(*Sensori di extra corsa + home + tastatori + presenza elemento nella pinza*)
MachinePalletizerModules.AX_X.IN.Px_Touch_1			 		:= Ok_sensores_Tastator OR (Re_In_TastatorePinza[1]  AND Re_In_TastatorePinza[2]) ;
MachinePalletizerModules.AX_X.IN.Px_Touch_2			 		:= Ok_sensores_Tastator OR ( Re_In_TastatorePinza[3]  AND Re_In_TastatorePinza[4]) ;
//MachinePalletizerModules.AX_X.IN.PX_TouchEmergency_1		:= I_TastatoreEmergenzaPinza_1 AND I_TastatoreEmergenzaPinza_2 AND I_TastatoreEmergenzaPinza_3 AND I_TastatoreEmergenzaPinza_4 OR NOT TouchErrorEnable;
MachinePalletizerModules.AX_X.IN.PX_TouchEmergency_1		:= (Re_In_TastatoreEmergenzaPinza[1] AND Re_In_TastatoreEmergenzaPinza[2])OR NOT TouchErrorEnable;
MachinePalletizerModules.AX_X.IN.PX_TouchEmergency_2		:= (Re_In_TastatoreEmergenzaPinza[3] AND Re_In_TastatoreEmergenzaPinza[4])OR NOT TouchErrorEnable;
MachinePalletizerModules.AX_X.IN.PX_GripPresence			:= NOT I_PHPresenzaMaterialePinza;
MachinePalletizerModules.AX_X.IN.Enable_TouchEmergency   	:= ADR(TouchErrorEnable);

MachinePalletizerModules.AX_X.Ax^.PxNegative 			:= NOT I_ExtraCorsaNegativo_X ;
MachinePalletizerModules.AX_X.Ax^.PxPositive 			:= NOT I_ExtraCorsaPositivo_X ;
IF MachinePalletizerModules.AX_X.AxHomingParameters^.InvertiDirezione THEN
	MachinePalletizerModules.AX_X.Ax^.PxHome 			:= NOT I_ExtraCorsaPositivo_X;
ELSE
	MachinePalletizerModules.AX_X.Ax^.PxHome 			:= NOT I_ExtraCorsaNegativo_X;
END_IF

MachinePalletizerModules.AX_X.Ax^.PxNegativeEnable 		:= TRUE;
MachinePalletizerModules.AX_X.Ax^.PxPositiveEnable 		:= TRUE;
MachinePalletizerModules.AX_X.Ax^.HomeExecutedAlwaysOn 	:= TRUE;
MachinePalletizerModules.AX_X.Ax^.DriveNeedReset 		:= DriveNeedReset;

MachinePalletizerModules.AX_X.Ax^.Parameter.MAXPosition 			:= AxisPar_X.MaxPosition;
MachinePalletizerModules.AX_X.Ax^.Parameter.MinPosition 			:= AxisPar_X.MinPosition;
MachinePalletizerModules.AX_X.Ax^.Parameter.HomeLagError			:= 0;
MachinePalletizerModules.AX_X.Ax^.EnableAutoWritePositionLimit 		:= TRUE;
(* Varie Modulo*)
MachinePalletizerModules.AX_X.AxisPar 					:= ADR(AxisPar_X);
MachinePalletizerModules.AX_X.ManCmd					:= ADR(ManCmd.X);
MachinePalletizerModules.AX_X.Cfg.TimeBase 				:= TimeBase;
MachinePalletizerModules.AX_X.Programma					:= ADR(ProgrammaToModule_X);


//@@@@@@@@@@@@@@@@@@@@@@@@@@@@@@@@@@@@@@@@@@@@@@@@@@@@@@@@@@@@@@@@@@@@@@@@@@@@@@@
ProgramaEjes.EjeX := ProgrammaToModule_X.ID ;
ProgramaEjes.CoordenadaEjeX := ProgrammaToModule_X.Quota_Destinazione ;
//@@@@@@@@@@@@@@@@@@@@@@@@@@@@@@@@@@@@@@@@@@@@@@@@@@@@@@@@@@@@@@@@@@@@@@@@@@@@@@
EncoderEsternoAsse_X.Pronto								:= I_EncoderX_Pronto;
MachinePalletizerModules.AX_X.EncoderEsterno			:= ADR(EncoderEsternoAsse_X);

(*AGGIORNAMENTO STATO DEL PROGEMMA IN ESECUZIONE*)
Programma_X[ProgrammaToModule_X.ID].Stato := ProgrammaToModule_X.Stato;
(************************************************************************
******************************* MODULO Y ********************************
************************************************************************)
(* Configurazione Asse Y *)
MachinePalletizerModules.AX_Y.Ax 							:= ADR(Y_AxisLib);
MachinePalletizerModules.AX_Y.Ax^.AxRef 					:= ADR(Y_Axis);
MachinePalletizerModules.AX_Y.Ax^.TimeBase 					:= TimeBase;
MachinePalletizerModules.AX_Y.Ax^.PowerEnable 				:= PowerEnableAssi;
MachinePalletizerModules.AX_Y.Ax^.PowerEnablePositive    	:= PowerEnableAssi AND (I_ExtraCorsaPositivo_Y OR NOT TouchErrorEnable);
MachinePalletizerModules.AX_Y.Ax^.PowerEnableNegative    	:= PowerEnableAssi AND (I_ExtraCorsaNegativo_Y OR NOT TouchErrorEnable);
MachinePalletizerModules.AX_Y.Ax^.EncoderType				:= ABSOLUTE_ENCODER;
MachinePalletizerModules.AX_Y.AxHomingParameters			:= ADR(AxisHomingParameters_Y);

(*Sensori di extra corsa + home + tastatori + presenza elemento nella pinza + sicurezza cinghia*)
MachinePalletizerModules.AX_Y.IN.BeltSafety				:= I_SicurezzaCinghia_Y OR NOT TouchErrorEnable;
MachinePalletizerModules.AX_Y.IN.Px_Touch_1			 	:= Ok_sensores_Tastator OR (Re_In_TastatorePinza[1]  AND Re_In_TastatorePinza[2]) ;
MachinePalletizerModules.AX_Y.IN.Px_Touch_2			 	:= Ok_sensores_Tastator OR (Re_In_TastatorePinza[3]  AND Re_In_TastatorePinza[4]) ;
//MachinePalletizerModules.AX_Y.IN.PX_TouchEmergency_1		:= I_TastatoreEmergenzaPinza_1 AND I_TastatoreEmergenzaPinza_2 AND I_TastatoreEmergenzaPinza_3 AND I_TastatoreEmergenzaPinza_4 OR NOT TouchErrorEnable;
MachinePalletizerModules.AX_Y.IN.PX_TouchEmergency_1		:= (Re_In_TastatoreEmergenzaPinza[1] AND Re_In_TastatoreEmergenzaPinza[2]) OR NOT TouchErrorEnable;
MachinePalletizerModules.AX_Y.IN.PX_TouchEmergency_2		:= ( Re_In_TastatoreEmergenzaPinza[3] AND Re_In_TastatoreEmergenzaPinza[4] )OR NOT TouchErrorEnable;;
MachinePalletizerModules.AX_Y.IN.PX_GripPresence			:= NOT I_PHPresenzaMaterialePinza;
MachinePalletizerModules.AX_Y.IN.Enable_TouchEmergency   := ADR(TouchErrorEnable);
MachinePalletizerModules.AX_Y.IN.SimulazioneSenzaHW		:= FALSE;//TEST_ENABLE;
MachinePalletizerModules.AX_Y.AbilitaOffsetInUscitaTasteggio   := TRUE;//FROM_HMI_PAL.HMI_AbilitaOffsetUscitaTasteggioPrelPallet;
MachinePalletizerModules.AX_Y.OffsetUscitaDaTasteggio	:=  HMI_OffsetUscitaTastatori;
MachinePalletizerModules.AX_Y.VelocitaDiUscitaDaTastatori := HMI_VelocitaDiUscitaDaTastatoriAxY;

MachinePalletizerModules.AX_Y.Ax^.PxNegative 			:= NOT I_ExtraCorsaNegativo_Y;
MachinePalletizerModules.AX_Y.Ax^.PxPositive 			:= NOT I_ExtraCorsaPositivo_Y;

IF MachinePalletizerModules.AX_Y.AxHomingParameters^.InvertiDirezione THEN
	MachinePalletizerModules.AX_Y.Ax^.PxHome 			:= NOT I_ExtraCorsaPositivo_Y;
ELSE
	MachinePalletizerModules.AX_Y.Ax^.PxHome 			:= NOT I_ExtraCorsaNegativo_Y;
END_IF

(* Varie Modulo*)
MachinePalletizerModules.AX_Y.Ax^.PxNegativeEnable 		:= TRUE;
MachinePalletizerModules.AX_Y.Ax^.PxPositiveEnable 		:= TRUE;
MachinePalletizerModules.AX_Y.Ax^.HomeExecutedAlwaysOn 	:= TRUE;
MachinePalletizerModules.AX_Y.Ax^.DriveNeedReset 		:= DriveNeedReset;

MachinePalletizerModules.AX_Y.Ax^.Parameter.MAXPosition 			:= AxisPar_Y.MaxPosition;
MachinePalletizerModules.AX_Y.Ax^.Parameter.MinPosition 			:= AxisPar_Y.MinPosition;
MachinePalletizerModules.AX_Y.Ax^.EnableAutoWritePositionLimit 		:= TRUE;
MachinePalletizerModules.AX_Y.Ax^.Parameter.HomeLagError			:= 0;

MachinePalletizerModules.AX_Y.AxisPar 					:= ADR(AxisPar_Y);
//MachinePalletizerModules.AX_Y.Status 					:= ADR(Status);
MachinePalletizerModules.AX_Y.ManCmd					:= ADR(ManCmd.Y);
MachinePalletizerModules.AX_Y.Cfg.TimeBase 				:= TimeBase;
MachinePalletizerModules.AX_Y.Programma					:= ADR(ProgrammaToModule_Y);

//@@@@@@@@@@@@@@@@@@@@@@@@@@@@@@@@@@@@@@@@@@@@@@@@@@@@@@@@@@
ProgramaEjes.EjeY := ProgrammaToModule_Y.ID;
ProgramaEjes.CoordenadaEjeY := ProgrammaToModule_Y.Quota_Destinazione;
//@@@@@@@@@@@@@@@@@@@@@@@@@@@@@@@@@@@@@@@@@@@@@@@@@@@@@@@@@@

//MachinePalletizerModules.AX_Y.ProgrammaNEXT				:= ADR(ProgrammaToModuleNEXT_Y);
(*AGGIORNAMENTO STATO DEL PROGEMMA IN ESECUZIONE*)
Programma_Y[ProgrammaToModule_Y.ID].Stato := ProgrammaToModule_Y.Stato;
//Programma_Y[ProgrammaToModuleNEXT_Y.ID].Stato := ProgrammaToModuleNEXT_Y.Stato;
(************************************************************************
******************************* MODULO Z ********************************
************************************************************************)
(* Configurazione Asse Z *)
MachinePalletizerModules.AX_Z.Ax 						:= ADR(Z_AxisLib);
MachinePalletizerModules.AX_Z.Ax^.AxRef 					:= ADR(Z_Axis);
MachinePalletizerModules.AX_Z.Ax^.TimeBase 				:= TimeBase;
MachinePalletizerModules.AX_Z.Ax^.PowerEnable 			:= PowerEnableAssi;
MachinePalletizerModules.AX_Z.Ax^.PowerEnablePositive    := PowerEnableAssi AND (I_ExtraCorsaPositivo_Z OR NOT TouchErrorEnable)AND (I_FermoSicurezzaRilasciato OR I_StartCicloPal);
//MachinePalletizerModules.AX_Z.Ax^.PowerEnableNegative    := PowerEnableAssi AND (I_ExtraCorsaNegativo_Z AND (I_TastatoreEmergenzaPinza_1 AND I_TastatoreEmergenzaPinza_2) OR NOT TouchErrorEnable) AND (I_FermoSicurezzaRilasciato OR I_StartCicloPal);
MachinePalletizerModules.AX_Z.Ax^.PowerEnableNegative    := PowerEnableAssi 
																AND (I_ExtraCorsaNegativo_Z AND (Re_In_TastatoreEmergenzaPinza[1] AND Re_In_TastatoreEmergenzaPinza[1]) 
																			OR NOT TouchErrorEnable) AND (I_FermoSicurezzaRilasciato OR I_StartCicloPal);
MachinePalletizerModules.AX_Z.Ax^.EncoderType			:= ABSOLUTE_ENCODER;
MachinePalletizerModules.AX_Z.AxHomingParameters			:= ADR(AxisHomingParameters_Z);

MachinePalletizerModules.AX_Z.Ax^.BrakePresent := false;//TRUE;
MachinePalletizerModules.AX_Z.Ax^.BrakeEnable  := FALSE;//TRUE;
MachinePalletizerModules.AX_Z.Ax^.Parameter.TimeBrakeOff := 200;
MachinePalletizerModules.AX_Z.Ax^.Parameter.TimeBrakeOn  := 200;
MachinePalletizerModules.AX_Z.Ax^.Parameter.TimeBrakeActivation := 60000;


(*Sensori di extra corsa + home + tastatori + presenza elemento nella pinza + sicurezza cinghia*)
MachinePalletizerModules.AX_Z.IN.BeltSafety				:= I_SicurezzaCinghia_Z OR NOT TouchErrorEnable;	

(* Gestione dei tastatori in base al tipo di prelievo ovvero all'elemento che è presente in prelievo *)
MachinePalletizerModules.AX_Z.ByPassTastatoriInUscitaTasteggio 	:= FALSE;
MachinePalletizerModules.AX_Z.InterventoPxASpazio				:= FALSE;
MachinePalletizerModules.AX_Z.SpazioInteventoPX					:= HMI_SpazioInterventoTastoriCartone;

MachinePalletizerModules.AX_Z.IN.Px_Touch_1			 		:= Ok_sensores_Tastator OR (Re_In_TastatorePinza[1]  AND Re_In_TastatorePinza[2]) ;
MachinePalletizerModules.AX_Z.IN.Px_Touch_2			 		:= Ok_sensores_Tastator OR (Re_In_TastatorePinza[3]  AND Re_In_TastatorePinza[4]) ;
//MachinePalletizerModules.AX_Z.IN.PX_TouchEmergency_1		:= I_TastatoreEmergenzaPinza_1 AND I_TastatoreEmergenzaPinza_2 AND I_TastatoreEmergenzaPinza_3 AND I_TastatoreEmergenzaPinza_4 OR NOT TouchErrorEnable;
MachinePalletizerModules.AX_Z.IN.PX_TouchEmergency_1		:= (Re_In_TastatoreEmergenzaPinza[1] AND Re_In_TastatoreEmergenzaPinza[2] ) OR NOT TouchErrorEnable;
MachinePalletizerModules.AX_Z.IN.PX_TouchEmergency_2		:= (Re_In_TastatoreEmergenzaPinza[3] AND Re_In_TastatoreEmergenzaPinza[4]) OR NOT TouchErrorEnable;;
MachinePalletizerModules.AX_Z.IN.PX_GripPresence			:= NOT I_PHPresenzaMaterialePinza;
MachinePalletizerModules.AX_Z.IN.Enable_TouchEmergency   	:= ADR(TouchErrorEnable);
MachinePalletizerModules.AX_Z.IN.SimulazioneSenzaHW			:= FALSE;//TEST_ENABLE;
(* Gestione Tasteggio *)
MachinePalletizerModules.AX_Z.AbilitaOffsetInUscitaTasteggio   := TRUE;//FROM_HMI_PAL.HMI_AbilitaOffsetUscitaTasteggioPrelPallet;
MachinePalletizerModules.AX_Z.OffsetUscitaDaTasteggio		:= HMI_OffsetUscitaTastatori;
MachinePalletizerModules.AX_Z.VelocitaDiUscitaDaTastatori 	:= HMI_VelocitaDiUscitaDaTastatoriAxZ;
MachinePalletizerModules.AX_Z.TempoRisalitaTastatori 		:= HMI_TempoPresaPiastrella;

MachinePalletizerModules.AX_Z.Ax^.PxNegative 			:= NOT I_ExtraCorsaNegativo_Z;
MachinePalletizerModules.AX_Z.Ax^.PxPositive 			:= NOT I_ExtraCorsaPositivo_Z;
IF MachinePalletizerModules.AX_Z.AxHomingParameters^.InvertiDirezione THEN
	MachinePalletizerModules.AX_Z.Ax^.PxHome 				:= NOT I_ExtraCorsaPositivo_Z;
ELSE
	MachinePalletizerModules.AX_Z.Ax^.PxHome 				:= NOT I_ExtraCorsaNegativo_Z;
END_IF
(* Varie Modulo*)
MachinePalletizerModules.AX_Z.Ax^.PxNegativeEnable 		:= TRUE;//NOT TEST_ENABLE;
MachinePalletizerModules.AX_Z.Ax^.PxPositiveEnable 		:= TRUE;//NOT TEST_ENABLE;
MachinePalletizerModules.AX_Z.Ax^.HomeExecutedAlwaysOn 	:= TRUE;
MachinePalletizerModules.AX_Z.Ax^.DriveNeedReset 		:= DriveNeedReset;//NOT TEST_ENABLE;

MachinePalletizerModules.AX_Z.Ax^.Parameter.HomeInvertDirection 	:= TRUE;
MachinePalletizerModules.AX_Z.Ax^.Parameter.MAXPosition 			:= AxisPar_Z.MaxPosition;
MachinePalletizerModules.AX_Z.Ax^.Parameter.MinPosition 			:= AxisPar_Z.MinPosition;
MachinePalletizerModules.AX_Z.Ax^.EnableAutoWritePositionLimit 	:= TRUE;
MachinePalletizerModules.AX_Z.Ax^.Parameter.HomeLagError			:= 0;

MachinePalletizerModules.AX_Z.AxisPar 					:= ADR(AxisPar_Z);
//MachinePalletizerModules.AX_Z.Status 					:= ADR(Status);
MachinePalletizerModules.AX_Z.ManCmd						:= ADR(ManCmd.Z);
MachinePalletizerModules.AX_Z.Cfg.TimeBase 				:= TimeBase;
MachinePalletizerModules.AX_Z.Programma					:= ADR(ProgrammaToModule_Z);
//@@@@@@@@@@@@@@@@@@@@@@@@@@@@@@@@@@@@@@@@@@@@@@@@@@@@@@@@@@
ProgramaEjes.EjeZ := ProgrammaToModule_Z.ID;
ProgramaEjes.CoordenadaEjeZ := ProgrammaToModule_Z.Quota_Destinazione;
//@@@@@@@@@@@@@@@@@@@@@@@@@@@@@@@@@@@@@@@@@@@@@@@@@@@@@@@@@@

//MachinePalletizerModules.AX_Z.ProgrammaNEXT				:= ADR(ProgrammaToModuleNEXT_Z);

(*AGGIORNAMENTO STATO DEL PROGEMMA IN ESECUZIONE*)
Programma_Z[ProgrammaToModule_Z.ID].Stato := ProgrammaToModule_Z.Stato;
//Programma_Z[ProgrammaToModuleNEXT_Z.ID].Stato := ProgrammaToModuleNEXT_Z.Stato;

(************************************************************************
******************************* MODULO J ********************************
************************************************************************)
(* Configurazione Asse J *)
MachinePalletizerModules.AX_J.Ax 						:= ADR(J_AxisLib);
MachinePalletizerModules.AX_J.Ax^.AxRef 				:= ADR(J_Axis);
MachinePalletizerModules.AX_J.Ax^.TimeBase 				:= TimeBase;
MachinePalletizerModules.AX_J.AxisPar 					:= ADR(AxisPar_J);
//MachinePalletizerModules.AX_J.Status 					:= ADR(Status);
MachinePalletizerModules.AX_J.ManCmd					:= ADR(ManCmd.J);
MachinePalletizerModules.AX_J.Cfg.TimeBase 				:= TimeBase;
MachinePalletizerModules.AX_J.Programma					:= ADR(ProgrammaToModule_J);
//@@@@@@@@@@@@@@@@@@@@@@@@@@@@@@@@@@@@@@@@@@@@@@@@@@@@@@@@@@
ProgramaEjes.EjeJ := ProgrammaToModule_J.ID;
ProgramaEjes.CoordenadaEjeJ := ProgrammaToModule_J.Quota_Destinazione;

//@@@@@@@@@@@@@@@@@@@@@@@@@@@@@@@@@@@@@@@@@@@@@@@@@@@@@@@@@@
(*RetardoAlarTastatore(IN := NOT I_TastatoreEmergenzaPinza_1 OR NOT I_TastatoreEmergenzaPinza_2 
							OR NOT I_TastatoreEmergenzaPinza_3 OR NOT I_TastatoreEmergenzaPinza_4 ,Pt:=T#30MS);*)
							
							

(*Sensori di extra corsa + home + tastatori + presenza elemento nella pinza*)
MachinePalletizerModules.AX_J.IN.Px_Touch_1			 	:=  Ok_sensores_Tastator OR (Re_In_TastatorePinza[1]  AND Re_In_TastatorePinza[2]) ;
MachinePalletizerModules.AX_J.IN.Px_Touch_2			 	:=  Ok_sensores_Tastator OR (Re_In_TastatorePinza[3]  AND Re_In_TastatorePinza[4]) ;
MachinePalletizerModules.AX_J.IN.PX_TouchEmergency_1	:= (Re_In_TastatoreEmergenzaPinza[1] AND Re_In_TastatoreEmergenzaPinza[2] ) OR NOT TouchErrorEnable;
MachinePalletizerModules.AX_J.IN.PX_TouchEmergency_2	:= (Re_In_TastatoreEmergenzaPinza[3] AND Re_In_TastatoreEmergenzaPinza[4] ) OR NOT TouchErrorEnable;;
MachinePalletizerModules.AX_J.AxHomingParameters		:= ADR(AxisHomingParameters_J);
MachinePalletizerModules.AX_J.Ax^.EncoderType			:= ABSOLUTE_ENCODER;
                                                        
MachinePalletizerModules.AX_J.IN.PX_GripPresence		:= NOT I_PHPresenzaMaterialePinza;
MachinePalletizerModules.AX_J.IN.Enable_TouchEmergency  := ADR(TouchErrorEnable);
MachinePalletizerModules.AX_J.IN.SimulazioneSenzaHW		:= FALSE;//TEST_ENABLE;

MachinePalletizerModules.AX_J.Ax^.TimeBase 				:= TimeBase;
MachinePalletizerModules.AX_J.Ax^.PowerEnable 			:= PowerEnableAssi;
MachinePalletizerModules.AX_J.Ax^.Parameter.HomeInvertDirection 	:= MachinePalletizerModules.AX_J.AxHomingParameters^.InvertiDirezione;
IF MachinePalletizerModules.AX_J.AxHomingParameters^.InvertiDirezione THEN
	MachinePalletizerModules.AX_J.Ax^.PxHome 			:= NOT I_ExtraCorsaPositivo_J;
ELSE
	MachinePalletizerModules.AX_J.Ax^.PxHome 			:= NOT I_ExtraCorsaNegativo_J;
END_IF
MachinePalletizerModules.AX_J.Ax^.PxNegative 			:= NOT I_ExtraCorsaNegativo_J;
MachinePalletizerModules.AX_J.Ax^.PxPositive 			:= NOT I_ExtraCorsaPositivo_J;

MachinePalletizerModules.AX_J.Ax^.PowerEnablePositive    := PowerEnableAssi AND (I_ExtraCorsaPositivo_J OR NOT TouchErrorEnable);
MachinePalletizerModules.AX_J.Ax^.PowerEnableNegative    := PowerEnableAssi AND (I_ExtraCorsaNegativo_J OR NOT TouchErrorEnable);

(* Varie Modulo*)
MachinePalletizerModules.AX_J.Ax^.PxNegativeEnable 		:= TRUE;
MachinePalletizerModules.AX_J.Ax^.PxPositiveEnable 		:= TRUE;//NOT TEST_ENABLE;
MachinePalletizerModules.AX_J.Ax^.HomeExecutedAlwaysOn 	:= TRUE;
MachinePalletizerModules.AX_J.Ax^.DriveNeedReset 		:= DriveNeedReset;//NOT TEST_ENABLE;

MachinePalletizerModules.AX_J.Ax^.Parameter.MAXPosition 			:= AxisPar_J.MaxPosition;
MachinePalletizerModules.AX_J.Ax^.Parameter.MinPosition 			:= AxisPar_J.MinPosition;
MachinePalletizerModules.AX_J.Ax^.EnableAutoWritePositionLimit 		:= TRUE;
MachinePalletizerModules.AX_J.Ax^.Parameter.HomeLagError			:= 0;
//FTC TASTEGGIO
MachinePalletizerModules.AX_J.IN_Pinza.InKeyence0_Byte0		:= I_Keyence180_Byte0;
MachinePalletizerModules.AX_J.IN_Pinza.InKeyence0_Byte1		:= I_Keyence180_Byte1;
MachinePalletizerModules.AX_J.IN_Pinza.InKeyence180_Byte0	:= I_Keyence0_Byte0; 
MachinePalletizerModules.AX_J.IN_Pinza.InKeyence180_Byte1	:= I_Keyence0_Byte1;

(*AGGIORNAMENTO STATO DEL PROGEMMA IN ESECUZIONE*)
Programma_J[ProgrammaToModule_J.ID].Stato := ProgrammaToModule_J.Stato;

{region " PINZA "}
(************************************************************************
***************** MODULO PINZA CON GESTIONE ASPIRAZIONI VARIE *************************
************************************************************************)
MachinePalletizerModules.Pinza.IN.TastoreCartoneDX	 			:= I_TastoreCartone1;
MachinePalletizerModules.Pinza.IN.TastoreCartoneSX	 			:= I_TastoreCartone2;
MachinePalletizerModules.Pinza.IN.ExtraCorsaPinzaSganciata 		:= I_ExtraCorsaPinzaSganciata;
MachinePalletizerModules.Pinza.IN.InKeyence0_Byte0				:= I_Keyence0_Byte0;
MachinePalletizerModules.Pinza.IN.InKeyence0_Byte1				:= I_Keyence0_Byte1;
MachinePalletizerModules.Pinza.IN.InKeyence180_Byte0			:= I_Keyence180_Byte0; 
MachinePalletizerModules.Pinza.IN.InKeyence180_Byte1			:= I_Keyence180_Byte1;

MachinePalletizerModules.Pinza.IN.InKeyence0_Byte0_2			:= I_Keyence0_Byte0_2;
MachinePalletizerModules.Pinza.IN.InKeyence0_Byte1_2			:= I_Keyence0_Byte1_2;
MachinePalletizerModules.Pinza.IN.InKeyence180_Byte0_2			:= I_Keyence180_Byte0_2; 
MachinePalletizerModules.Pinza.IN.InKeyence180_Byte1_2			:= I_Keyence180_Byte1_2;
			   
MachinePalletizerModules.Pinza.ManCmd							:= ADR(ManCmd.Pinza);
MachinePalletizerModules.Pinza.Cfg.TimeBase 					:= TimeBase;
MachinePalletizerModules.Pinza.ModuleJ							:= ADR(MachinePalletizerModules.AX_J);
MachinePalletizerModules.Pinza.Mission							:= ADR(Mission);

(* Cilindro Apertura *)
MachinePalletizerModules.Pinza.CilindroApertura 									:= ADR(CilindroAperturaPinza);
MachinePalletizerModules.Pinza.CilindroApertura^.Enable_RUN 						:= EnablePneumatica;	
MachinePalletizerModules.Pinza.CilindroApertura^.Config.ForceActive_OnStartup 		:= FALSE;				// Se a Startup il cilindro è in stato non definito forza Inattivo (CONFIG)	
MachinePalletizerModules.Pinza.CilindroApertura^.Config.ForceInactive_OnStartup 	:= TRUE;				// Se a Startup il cilindro è in stato non definito forza Attivo (CONFIG)
MachinePalletizerModules.Pinza.CilindroApertura^.Config.TimeBase 					:= Timebase;							// Base dei tempi
MachinePalletizerModules.Pinza.CilindroApertura^.Parameter.ActivationTime 			:= 100;						// [ms] di Attivazione/Timeout (PARAMETRO)
MachinePalletizerModules.Pinza.CilindroApertura^.Parameter.DeactivationTime 		:= 100;						// [ms] di Disattivazione/Timeout (PARAMETRO)
MachinePalletizerModules.Pinza.CilindroApertura^.Parameter.FeedbackType 			:= DEVICE_WITHOUT_FEEDBACK; 	// Scelta dei reed presenti
MachinePalletizerModules.Pinza.CilindroApertura^.Parameter.PxActive_FilterTime_OFF 	:= 0;					// [ms] di filtro sensore Attivo ON (0=NO filtro) (PARAMETRO)
MachinePalletizerModules.Pinza.CilindroApertura^.Parameter.PxActive_FilterTime_ON 	:= 0;					// [ms] di filtro sensore Attivo OFF (0=NO filtro) (PARAMETRO)
MachinePalletizerModules.Pinza.CilindroApertura^.Parameter.PxInactive_FilterTime_OFF 	:= 0;				// [ms] di filtro sensore Inattivo ON (0=NO filtro) (PARAMETRO)
MachinePalletizerModules.Pinza.CilindroApertura^.Parameter.PxInactive_FilterTime_ON 	:= 0;				// [ms] di filtro sensore Inattivo ON (0=NO filtro) (PARAMETRO)
MachinePalletizerModules.Pinza.CilindroApertura^.Parameter.PxLatchFunction_Enable 	:= TRUE;				// Enable gestione sensori con latch (PARAMETRO)
MachinePalletizerModules.Pinza.CilindroApertura^.IN.PX_Active 						:= I_PinzaApertaDX AND I_PinzaApertaSX;	// IN sensore aperto
MachinePalletizerModules.Pinza.CilindroApertura^.IN.PX_Inactive 					:= I_PinzaChiusaDX AND I_PinzaChiusaSX; // IN sensore chiuso	
MachinePalletizerModules.Pinza.IN.FTC_FaldaDX										:= I_PHPresenzaFaldaDX;
MachinePalletizerModules.Pinza.IN.FTC_FaldaSX										:= I_PHPresenzaFaldaSX;
MachinePalletizerModules.Pinza.AbilitaAperturaAutomaticaPinza						:= HMI_AbilitaAperturaAutomaticaPinza;
			   
(* OVEM ventose DX *)	
MachinePalletizerModules.Pinza.AspirazioneDX1 							:= ADR(Ovem1);
MachinePalletizerModules.Pinza.AspirazioneDX1^.IN.LivelloDepressione 	:=  (SHL(I_LivelloDepressioneOVEM_BH_1,8) OR I_LivelloDepressioneOVEM_BL_1) ;
(* Ingressi Ovem *)
MachinePalletizerModules.Pinza.AspirazioneDX1^.IN.PortQualifier		:=  I_PortQualifierOVEM_1;
MachinePalletizerModules.Pinza.AspirazioneDX1^.IN.TimeStamp			:=  I_TimeStampCiabattaPinzaK515;
MachinePalletizerModules.Pinza.AspirazioneDX1^.IN.AirOK				:=  I_AriaOK;
(* Comunicazione OVEM *)
ComunicazioneOvem1.sNetId 												:= F_CreateAmsNetId(I_CiabattaPinzaK515AMSADDR.netId);
ComunicazioneOvem1.nSlaveAddr 											:= I_CiabattaPinzaK515AMSADDR.port;
ComunicazioneOvem1.nPorta 												:= 1;
MachinePalletizerModules.Pinza.AspirazioneDX1^.IN_Comunication			:= ADR(ComunicazioneOvem1);
(* COMANDI *)
MachinePalletizerModules.Pinza.AspirazioneDX1^.Command					:= ADR(CommandOVEM_1);
(* PARAMETRI *)
FROM_HMI_PAL.HMI_OvemParameters.SogliaDepressione_1B 	:= FROM_HMI_PAL.HMI_OvemParameters.SogliaDepressione_1;
FROM_HMI_PAL.HMI_OvemParameters.SogliaDepressione_2 	:= FROM_HMI_PAL.HMI_OvemParameters.SogliaDepressione_1;
FROM_HMI_PAL.HMI_OvemParameters.SogliaDepressione_2B 	:= FROM_HMI_PAL.HMI_OvemParameters.SogliaDepressione_1;
IF (FROM_HMI_PAL.HMI_OvemParameters.SogliaDepressione_1 - FROM_HMI_PAL.HMI_OvemParameters.IsteresiDepressione_1) <= 0 THEN //Se l'isteresi è >= della soglia, la forzo a zero
	FROM_HMI_PAL.HMI_OvemParameters.IsteresiDepressione_1 := 0;
END_IF

MachinePalletizerModules.Pinza.AspirazioneDX1^.Parameters.TempoInvioComandiCoe					:= 40;
MachinePalletizerModules.Pinza.AspirazioneDX1^.IN_TargetParameters								:= FROM_HMI_PAL.HMI_OvemParameters;
MachinePalletizerModules.Pinza.AspirazioneDX1^.Parameters.AbilitaScritturaAutomaticaParametri 	:= TRUE;
MachinePalletizerModules.Pinza.AspirazioneDX1^.Parameters.UtilizzaStatoDepressione_OVEM 		:= TRUE;
MachinePalletizerModules.Pinza.AspirazioneDX1^.Parameters.TimeDepLOST						:= 200;
MachinePalletizerModules.Pinza.AspirazioneDX1^.Parameters.TimeDepOK							:= 100;
MachinePalletizerModules.Pinza.AspirazioneDX1^.Parameters.TipoSoffio							:= 1;//Soffio Automatico e gestito dall'ovem
MachinePalletizerModules.Pinza.AspirazioneDX1^.Parameters.AbilitaCalcoloAutoSoglia			:= TRUE;
MachinePalletizerModules.Pinza.AspirazioneDX1^.Parameters.TipologiaOvem						:= 1;//Ovem di tipo NO
(* OVEM ventose SX *)
MachinePalletizerModules.Pinza.AspirazioneSX1 							:= ADR(Ovem2);
MachinePalletizerModules.Pinza.AspirazioneSX1^.IN.LivelloDepressione 	:=  (SHL(I_LivelloDepressioneOVEM_BH_2,8) OR I_LivelloDepressioneOVEM_BL_2) ;
(* Ingressi Ovem *)
MachinePalletizerModules.Pinza.AspirazioneSX1^.IN.PortQualifier		:=  I_PortQualifierOVEM_2;
MachinePalletizerModules.Pinza.AspirazioneSX1^.IN.TimeStamp			:=  I_TimeStampCiabattaPinzaK516;
MachinePalletizerModules.Pinza.AspirazioneSX1^.IN.AirOK				:=  I_AriaOK;
(* Comunicazione OVEM *)
ComunicazioneOvem2.sNetId 													:= F_CreateAmsNetId(I_CiabattaPinzaK516AMSADDR.netId);
ComunicazioneOvem2.nSlaveAddr 												:= I_CiabattaPinzaK516AMSADDR.port;
ComunicazioneOvem2.nPorta 													:= 1;
MachinePalletizerModules.Pinza.AspirazioneSX1^.IN_Comunication			:= ADR(ComunicazioneOvem2);
(* COMANDI *)
MachinePalletizerModules.Pinza.AspirazioneSX1^.Command					:= ADR(CommandOVEM_2);
(* PARAMETRI *)
MachinePalletizerModules.Pinza.AspirazioneSX1^.Parameters := MachinePalletizerModules.Pinza.AspirazioneDX1^.Parameters;
MachinePalletizerModules.Pinza.AspirazioneSX1^.IN_TargetParameters := MachinePalletizerModules.Pinza.AspirazioneDX1^.IN_TargetParameters;

(* OVEM ventose DX2 *)	
MachinePalletizerModules.Pinza.AspirazioneDX2 							:= ADR(Ovem12);
MachinePalletizerModules.Pinza.AspirazioneDX2^.IN.LivelloDepressione 	:=  (SHL(I_LivelloDepressioneOVEM_BH_12,8) OR I_LivelloDepressioneOVEM_BL_12) ;
(* Ingressi Ovem *)
MachinePalletizerModules.Pinza.AspirazioneDX2^.IN.PortQualifier			:=  I_PortQualifierOVEM_12;
MachinePalletizerModules.Pinza.AspirazioneDX2^.IN.TimeStamp				:=  I_TimeStampCiabattaPinzaK515;
MachinePalletizerModules.Pinza.AspirazioneDX2^.IN.AirOK					:=  I_AriaOK;
(* Comunicazione OVEM *)
ComunicazioneOvem12.sNetId 												:= F_CreateAmsNetId(I_CiabattaPinzaK515AMSADDR.netId);
ComunicazioneOvem12.nSlaveAddr 											:= I_CiabattaPinzaK515AMSADDR.port;
ComunicazioneOvem12.nPorta 												:= 5;
MachinePalletizerModules.Pinza.AspirazioneDX2^.IN_Comunication			:= ADR(ComunicazioneOvem12);
(* COMANDI *)
MachinePalletizerModules.Pinza.AspirazioneDX2^.Command					:= ADR(CommandOVEM_12);
(* PARAMETRI *)
MachinePalletizerModules.Pinza.AspirazioneDX2^.Parameters 			:= MachinePalletizerModules.Pinza.AspirazioneDX1^.Parameters;
MachinePalletizerModules.Pinza.AspirazioneDX2^.IN_TargetParameters 	:= MachinePalletizerModules.Pinza.AspirazioneDX1^.IN_TargetParameters;

(* OVEM ventose SX2 *)
MachinePalletizerModules.Pinza.AspirazioneSX2 							:= ADR(Ovem22);
MachinePalletizerModules.Pinza.AspirazioneSX2^.IN.LivelloDepressione 	:=  (SHL(I_LivelloDepressioneOVEM_BH_22,8) OR I_LivelloDepressioneOVEM_BL_22) ;
(* Ingressi Ovem *)
MachinePalletizerModules.Pinza.AspirazioneSX2^.IN.PortQualifier		:=  I_PortQualifierOVEM_22;
MachinePalletizerModules.Pinza.AspirazioneSX2^.IN.TimeStamp			:=  I_TimeStampCiabattaPinzaK516;
MachinePalletizerModules.Pinza.AspirazioneSX2^.IN.AirOK				:=  I_AriaOK;
(* Comunicazione OVEM *)
ComunicazioneOvem22.sNetId 													:= F_CreateAmsNetId(I_CiabattaPinzaK516AMSADDR.netId);
ComunicazioneOvem22.nSlaveAddr 												:= I_CiabattaPinzaK516AMSADDR.port;
ComunicazioneOvem22.nPorta 													:= 2;
MachinePalletizerModules.Pinza.AspirazioneSX2^.IN_Comunication			:= ADR(ComunicazioneOvem22);
(* COMANDI *)
MachinePalletizerModules.Pinza.AspirazioneSX2^.Command					:= ADR(CommandOVEM_22);
(* PARAMETRI *)
MachinePalletizerModules.Pinza.AspirazioneSX2^.Parameters 			:= MachinePalletizerModules.Pinza.AspirazioneDX1^.Parameters;
MachinePalletizerModules.Pinza.AspirazioneSX2^.IN_TargetParameters 	:= MachinePalletizerModules.Pinza.AspirazioneDX1^.IN_TargetParameters;
						 
MachinePalletizerModules.Pinza.IN.ByPassSensoreVuoto := HMI_AbilitaSimulazioneAVuoto;

(* Cilindro Sblocco Pinza *)
MachinePalletizerModules.Pinza.CilindroSbloccoRotazione 									:= ADR(CilindroSbloccoPinza);
MachinePalletizerModules.Pinza.CilindroSbloccoRotazione^.Enable_RUN 						:= EnablePneumatica;	
MachinePalletizerModules.Pinza.CilindroSbloccoRotazione^.Config.ForceActive_OnStartup 		:= FALSE;				// Se a Startup il cilindro è in stato non definito forza Inattivo (CONFIG)	
MachinePalletizerModules.Pinza.CilindroSbloccoRotazione^.Config.ForceInactive_OnStartup 	:= TRUE;				// Se a Startup il cilindro è in stato non definito forza Attivo (CONFIG)
MachinePalletizerModules.Pinza.CilindroSbloccoRotazione^.Config.TimeBase 					:= Timebase;			// Base dei tempi
MachinePalletizerModules.Pinza.CilindroSbloccoRotazione^.Parameter.ActivationTime 			:= 1000;				// [ms] di Attivazione/Timeout (PARAMETRO)
MachinePalletizerModules.Pinza.CilindroSbloccoRotazione^.Parameter.DeactivationTime 		:= 2000;					// [ms] di Disattivazione/Timeout (PARAMETRO)
MachinePalletizerModules.Pinza.CilindroSbloccoRotazione^.Parameter.FeedbackType 			:= DEVICE_WITH_INACTIVE_FEEDBACK; 	// Scelta dei reed presenti
MachinePalletizerModules.Pinza.CilindroSbloccoRotazione^.Parameter.PxActive_FilterTime_OFF 	:= 0;				// [ms] di filtro sensore Attivo ON (0=NO filtro) (PARAMETRO)
MachinePalletizerModules.Pinza.CilindroSbloccoRotazione^.Parameter.PxActive_FilterTime_ON 	:= 0;				// [ms] di filtro sensore Attivo OFF (0=NO filtro) (PARAMETRO)
MachinePalletizerModules.Pinza.CilindroSbloccoRotazione^.Parameter.PxInactive_FilterTime_OFF 	:= 0;				// [ms] di filtro sensore Inattivo ON (0=NO filtro) (PARAMETRO)
MachinePalletizerModules.Pinza.CilindroSbloccoRotazione^.Parameter.PxInactive_FilterTime_ON 	:= 0;				// [ms] di filtro sensore Inattivo ON (0=NO filtro) (PARAMETRO)
MachinePalletizerModules.Pinza.CilindroSbloccoRotazione^.Parameter.PxLatchFunction_Enable 	:= TRUE;			// Enable gestione sensori con latch (PARAMETRO)
MachinePalletizerModules.Pinza.CilindroSbloccoRotazione^.IN.PX_Active 						:= FALSE;			// IN sensore Alto
MachinePalletizerModules.Pinza.CilindroSbloccoRotazione^.IN.PX_Inactive 					:= I_RotazioneColonnaBloccata;			// IN sensore Basso 	
MachinePalletizerModules.Pinza.AbilitazioneSbloccoRotazione									:= HMI_AbilitaSbloccoRotPinza;
(* Cilindro Sblocco Bascolante *)
MachinePalletizerModules.Pinza.CilindroSbloccoBascolante 									:= ADR(CilindroSbloccoBascolante);
MachinePalletizerModules.Pinza.CilindroSbloccoBascolante^.Enable_RUN 						:= EnablePneumatica;	
MachinePalletizerModules.Pinza.CilindroSbloccoBascolante^.Config.ForceActive_OnStartup 		:= FALSE;				// Se a Startup il cilindro è in stato non definito forza Inattivo (CONFIG)	
MachinePalletizerModules.Pinza.CilindroSbloccoBascolante^.Config.ForceInactive_OnStartup 	:= TRUE;				// Se a Startup il cilindro è in stato non definito forza Attivo (CONFIG)
MachinePalletizerModules.Pinza.CilindroSbloccoBascolante^.Config.TimeBase 					:= Timebase;			// Base dei tempi
MachinePalletizerModules.Pinza.CilindroSbloccoBascolante^.Parameter.ActivationTime 			:= 500;				// [ms] di Attivazione/Timeout (PARAMETRO)
MachinePalletizerModules.Pinza.CilindroSbloccoBascolante^.Parameter.DeactivationTime 		:= 500;					// [ms] di Disattivazione/Timeout (PARAMETRO)
MachinePalletizerModules.Pinza.CilindroSbloccoBascolante^.Parameter.FeedbackType 			:= DEVICE_WITH_INACTIVE_FEEDBACK; 	// Scelta dei reed presenti
MachinePalletizerModules.Pinza.CilindroSbloccoBascolante^.Parameter.ActivationTime 			:= 1000;
MachinePalletizerModules.Pinza.CilindroSbloccoBascolante^.Parameter.PxActive_FilterTime_OFF := 0;				// [ms] di filtro sensore Attivo ON (0=NO filtro) (PARAMETRO)
MachinePalletizerModules.Pinza.CilindroSbloccoBascolante^.Parameter.PxActive_FilterTime_ON 	:= 0;				// [ms] di filtro sensore Attivo OFF (0=NO filtro) (PARAMETRO)
MachinePalletizerModules.Pinza.CilindroSbloccoBascolante^.Parameter.PxInactive_FilterTime_OFF 	:= 0;				// [ms] di filtro sensore Inattivo ON (0=NO filtro) (PARAMETRO)
MachinePalletizerModules.Pinza.CilindroSbloccoBascolante^.Parameter.PxInactive_FilterTime_ON 	:= 0;				// [ms] di filtro sensore Inattivo ON (0=NO filtro) (PARAMETRO)
MachinePalletizerModules.Pinza.CilindroSbloccoBascolante^.Parameter.PxLatchFunction_Enable 	:= TRUE;			// Enable gestione sensori con latch (PARAMETRO)
MachinePalletizerModules.Pinza.CilindroSbloccoBascolante^.IN.PX_Active 						:= FALSE;			// IN sensore Alto
MachinePalletizerModules.Pinza.CilindroSbloccoBascolante^.IN.PX_Inactive 					:= I_BascolantePinzaBloccato;			// IN sensore Basso 	
MachinePalletizerModules.Pinza.AbilitazioneSbloccoBascolante								:= HMI_AbilitaBascolantePinza;
		  
(* Aspirazione Falda DX *)
MachinePalletizerModules.Pinza.AspirazioneFaldaDX										:= ADR(AspirazioneFaldaDX);
MachinePalletizerModules.Pinza.AspirazioneFaldaDX^.Enable_RUN 						:= EnablePneumatica;	
MachinePalletizerModules.Pinza.AspirazioneFaldaDX^.Config.ForceActive_OnStartup 		:= FALSE;				// Se a Startup il cilindro è in stato non definito forza Inattivo (CONFIG)	
MachinePalletizerModules.Pinza.AspirazioneFaldaDX^.Config.ForceInactive_OnStartup 	:= TRUE;				// Se a Startup il cilindro è in stato non definito forza Attivo (CONFIG)
MachinePalletizerModules.Pinza.AspirazioneFaldaDX^.Config.TimeBase 					:= Timebase;			// Base dei tempi
MachinePalletizerModules.Pinza.AspirazioneFaldaDX^.Parameter.ActivationTime 		:= 1;				// [ms] di Attivazione/Timeout (PARAMETRO)
MachinePalletizerModules.Pinza.AspirazioneFaldaDX^.Parameter.DeactivationTime 		:= 1;					// [ms] di Disattivazione/Timeout (PARAMETRO)
MachinePalletizerModules.Pinza.AspirazioneFaldaDX^.Parameter.FeedbackType 			:= DEVICE_WITHOUT_FEEDBACK; 	// Scelta dei reed presenti
MachinePalletizerModules.Pinza.AspirazioneFaldaDX^.Parameter.PxActive_FilterTime_OFF 	:= 0;					// [ms] di filtro sensore Attivo ON (0=NO filtro) (PARAMETRO)
MachinePalletizerModules.Pinza.AspirazioneFaldaDX^.Parameter.PxActive_FilterTime_ON 	:= 0;					// [ms] di filtro sensore Attivo OFF (0=NO filtro) (PARAMETRO)
MachinePalletizerModules.Pinza.AspirazioneFaldaDX^.Parameter.PxInactive_FilterTime_OFF 	:= 0;				// [ms] di filtro sensore Inattivo ON (0=NO filtro) (PARAMETRO)
MachinePalletizerModules.Pinza.AspirazioneFaldaDX^.Parameter.PxInactive_FilterTime_ON 	:= 0;				// [ms] di filtro sensore Inattivo ON (0=NO filtro) (PARAMETRO)
MachinePalletizerModules.Pinza.AspirazioneFaldaDX^.Parameter.PxLatchFunction_Enable 		:= TRUE;			// Enable gestione sensori con latch (PARAMETRO)
MachinePalletizerModules.Pinza.AspirazioneFaldaDX^.IN.PX_Active 							:= FALSE;			// IN sensore Alto
MachinePalletizerModules.Pinza.AspirazioneFaldaDX^.IN.PX_Inactive 						:= FALSE;			// IN sensore Basso 	
(* Aspirazione Falda SX *)
MachinePalletizerModules.Pinza.AspirazioneFaldaSX									:= ADR(AspirazioneFaldaSX);
MachinePalletizerModules.Pinza.AspirazioneFaldaSX^.Enable_RUN 						:= EnablePneumatica;	
MachinePalletizerModules.Pinza.AspirazioneFaldaSX^.Config.ForceActive_OnStartup 	:= FALSE;				// Se a Startup il cilindro è in stato non definito forza Inattivo (CONFIG)	
MachinePalletizerModules.Pinza.AspirazioneFaldaSX^.Config.ForceInactive_OnStartup 	:= TRUE;				// Se a Startup il cilindro è in stato non definito forza Attivo (CONFIG)
MachinePalletizerModules.Pinza.AspirazioneFaldaSX^.Config.TimeBase 					:= Timebase;			// Base dei tempi
MachinePalletizerModules.Pinza.AspirazioneFaldaSX^.Parameter.ActivationTime 		:= 1;				// [ms] di Attivazione/Timeout (PARAMETRO)
MachinePalletizerModules.Pinza.AspirazioneFaldaSX^.Parameter.DeactivationTime 		:= 1;					// [ms] di Disattivazione/Timeout (PARAMETRO)
MachinePalletizerModules.Pinza.AspirazioneFaldaSX^.Parameter.FeedbackType 			:= DEVICE_WITHOUT_FEEDBACK; 	// Scelta dei reed presenti
MachinePalletizerModules.Pinza.AspirazioneFaldaSX^.Parameter.PxActive_FilterTime_OFF 	:= 0;					// [ms] di filtro sensore Attivo ON (0=NO filtro) (PARAMETRO)
MachinePalletizerModules.Pinza.AspirazioneFaldaSX^.Parameter.PxActive_FilterTime_ON 	:= 0;					// [ms] di filtro sensore Attivo OFF (0=NO filtro) (PARAMETRO)
MachinePalletizerModules.Pinza.AspirazioneFaldaSX^.Parameter.PxInactive_FilterTime_OFF 	:= 0;				// [ms] di filtro sensore Inattivo ON (0=NO filtro) (PARAMETRO)
MachinePalletizerModules.Pinza.AspirazioneFaldaSX^.Parameter.PxInactive_FilterTime_ON 	:= 0;				// [ms] di filtro sensore Inattivo ON (0=NO filtro) (PARAMETRO)
MachinePalletizerModules.Pinza.AspirazioneFaldaSX^.Parameter.PxLatchFunction_Enable 		:= TRUE;			// Enable gestione sensori con latch (PARAMETRO)
MachinePalletizerModules.Pinza.AspirazioneFaldaSX^.IN.PX_Active 							:= FALSE;			// IN sensore Alto
MachinePalletizerModules.Pinza.AspirazioneFaldaSX^.IN.PX_Inactive 							:= FALSE;			// IN sensore Basso 	
	 

{endregion}

(* ******************************************************************************************************** *)
(* Machine/Modules Calls *)
(* ******************************************************************************************************** *)

MachinePalletizerGatesAccess.GateAccessConsolle.MachineCmd 					:= ADR(MachinePalletizer_TF.Cmd);
MachinepalletizerGatesAccess.GateAccessConsolle.MachineCmdExe 				:= ADR(MachinePalletizer_TF.CmdExe);
MachinepalletizerGatesAccess.GateAccessConsolle.MachineState 				:= ADR(MachinePalletizer_TF.State);
MachinepalletizerGatesAccess.GateAccessConsolle.MachineError 				:= ADR(MachinePalletizer_TF.Error);
MachinepalletizerGatesAccess.GateAccessConsolle.MachineMode 				:= ADR(MachinePalletizer_TF.IN.Mode);
MachinepalletizerGatesAccess.GateAccessConsolle.TimeBase 					:= TimeBase;
MachinepalletizerGatesAccess.GateAccessConsolle.AccessRequest				:= NOT I_RichiestaIngressoConsolle;
MachinepalletizerGatesAccess.GateAccessConsolle.AccessDone					:= I_ResetRichiestaIngressoConsolle;
MachinepalletizerGatesAccess.GateAccessConsolle.TilterPhaseStopDone			:= FALSE;
MachinepalletizerGatesAccess.GateAccessConsolle.PowerOK						:= I_MarciaOK;

MachinePalletizerGatesAccess.GateAccessPS306.MachineCmd 					:= ADR(MachinePalletizer_TF.Cmd);
MachinepalletizerGatesAccess.GateAccessPS306.MachineCmdExe 					:= ADR(MachinePalletizer_TF.CmdExe);
MachinepalletizerGatesAccess.GateAccessPS306.MachineState 					:= ADR(MachinePalletizer_TF.State);
MachinepalletizerGatesAccess.GateAccessPS306.MachineError 					:= ADR(MachinePalletizer_TF.Error);
MachinepalletizerGatesAccess.GateAccessPS306.MachineMode 					:= ADR(MachinePalletizer_TF.IN.Mode);
MachinepalletizerGatesAccess.GateAccessPS306.Modules 						:= ADR(MachinePalletizerModules);
MachinepalletizerGatesAccess.GateAccessPS306.Mission	 					:= ADR(Mission);
MachinepalletizerGatesAccess.GateAccessPS306.TimeBase 						:= TimeBase;
MachinepalletizerGatesAccess.GateAccessPS306.AccessRequest					:= NOT I_RichiestaIngressoPS306;
MachinepalletizerGatesAccess.GateAccessPS306.AccessDone						:= I_ResetRichiestaIngressoPS306;
MachinepalletizerGatesAccess.GateAccessPS306.TilterPhaseStopDone			:= FALSE;
MachinepalletizerGatesAccess.GateAccessPS306.PowerOK						:= I_MarciaOK;
MachinepalletizerGatesAccess.GateAccessPS306.MacchinaInLavoroZonaOpposta 	:= PortaleADx;


MachinePalletizerGatesAccess.GateAccessPS307.MachineCmd 					:= ADR(MachinePalletizer_TF.Cmd);
MachinepalletizerGatesAccess.GateAccessPS307.MachineCmdExe 					:= ADR(MachinePalletizer_TF.CmdExe);
MachinepalletizerGatesAccess.GateAccessPS307.MachineState 					:= ADR(MachinePalletizer_TF.State);
MachinepalletizerGatesAccess.GateAccessPS307.MachineError 					:= ADR(MachinePalletizer_TF.Error);
MachinepalletizerGatesAccess.GateAccessPS307.MachineMode 					:= ADR(MachinePalletizer_TF.IN.Mode);
MachinepalletizerGatesAccess.GateAccessPS307.Modules 						:= ADR(MachinePalletizerModules);
MachinepalletizerGatesAccess.GateAccessPS307.Mission	 					:= ADR(Mission);
MachinepalletizerGatesAccess.GateAccessPS307.TimeBase 						:= TimeBase;
MachinepalletizerGatesAccess.GateAccessPS307.AccessRequest					:= NOT I_RichiestaIngressoPS307;
MachinepalletizerGatesAccess.GateAccessPS307.AccessDone						:= I_ResetRichiestaIngressoPS307;
MachinepalletizerGatesAccess.GateAccessPS307.TilterPhaseStopDone			:= FALSE;
MachinepalletizerGatesAccess.GateAccessPS307.PowerOK						:= I_MarciaOK;
MachinepalletizerGatesAccess.GateAccessPS307.MacchinaInLavoroZonaOpposta 	:= PortaleADx;


MachinePalletizerGatesAccess.GateAccessPS308.MachineCmd 					:= ADR(MachinePalletizer_TF.Cmd);
MachinepalletizerGatesAccess.GateAccessPS308.MachineCmdExe 					:= ADR(MachinePalletizer_TF.CmdExe);
MachinepalletizerGatesAccess.GateAccessPS308.MachineState 					:= ADR(MachinePalletizer_TF.State);
MachinepalletizerGatesAccess.GateAccessPS308.MachineError 					:= ADR(MachinePalletizer_TF.Error);
MachinepalletizerGatesAccess.GateAccessPS308.MachineMode 					:= ADR(MachinePalletizer_TF.IN.Mode);
MachinepalletizerGatesAccess.GateAccessPS308.Modules 						:= ADR(MachinePalletizerModules);
MachinepalletizerGatesAccess.GateAccessPS308.Mission	 					:= ADR(Mission);
MachinepalletizerGatesAccess.GateAccessPS308.TimeBase 						:= TimeBase;
MachinepalletizerGatesAccess.GateAccessPS308.AccessRequest					:= NOT I_RichiestaIngressoPS308;
MachinepalletizerGatesAccess.GateAccessPS308.AccessDone						:= I_ResetRichiestaIngressoPS308;
MachinepalletizerGatesAccess.GateAccessPS308.TilterPhaseStopDone			:= FALSE;
MachinepalletizerGatesAccess.GateAccessPS308.PowerOK						:= I_MarciaOK;
MachinepalletizerGatesAccess.GateAccessPS308.MacchinaInLavoroZonaOpposta 	:= PortaleASx;


MachinePalletizerGatesAccess.GateAccessPS309.MachineCmd 					:= ADR(MachinePalletizer_TF.Cmd);
MachinepalletizerGatesAccess.GateAccessPS309.MachineCmdExe 					:= ADR(MachinePalletizer_TF.CmdExe);
MachinepalletizerGatesAccess.GateAccessPS309.MachineState 					:= ADR(MachinePalletizer_TF.State);
MachinepalletizerGatesAccess.GateAccessPS309.MachineError 					:= ADR(MachinePalletizer_TF.Error);
MachinepalletizerGatesAccess.GateAccessPS309.MachineMode 					:= ADR(MachinePalletizer_TF.IN.Mode);
MachinepalletizerGatesAccess.GateAccessPS309.Modules 						:= ADR(MachinePalletizerModules);
MachinepalletizerGatesAccess.GateAccessPS309.Mission	 					:= ADR(Mission);
MachinepalletizerGatesAccess.GateAccessPS309.TimeBase 						:= TimeBase;
MachinepalletizerGatesAccess.GateAccessPS309.AccessRequest					:= NOT I_RichiestaIngressoPS309;
MachinepalletizerGatesAccess.GateAccessPS309.AccessDone						:= I_ResetRichiestaIngressoPS309;
MachinepalletizerGatesAccess.GateAccessPS309.TilterPhaseStopDone			:= FALSE;
MachinepalletizerGatesAccess.GateAccessPS309.PowerOK						:= I_MarciaOK;
MachinepalletizerGatesAccess.GateAccessPS309.MacchinaInLavoroZonaOpposta 	:= PortaleASx;


MachinePalletizer_TF();
MachinepalletizerGatesAccess.GateAccessConsolle();
MachinepalletizerGatesAccess.GateAccessPS306();
MachinepalletizerGatesAccess.GateAccessPS307();
MachinepalletizerGatesAccess.GateAccessPS308();
MachinepalletizerGatesAccess.GateAccessPS309();
MachinePalletizerModules.AX_X();
MachinePalletizerModules.AX_Y();
MachinePalletizerModules.AX_Z();
MachinePalletizerModules.AX_J();
MachinePalletizerModules.Pinza();

(* Valutazione Input Safety *)
ResetNecessarioCentralinaSafety := I_SafetyCOMERR OR I_SafetyFBERR OR I_SafetyOTHERERR OR I_SafetyOUTERR OR
									I_SafetyCOMERR2 OR I_SafetyFBERR2 OR I_SafetyOTHERERR2 OR I_SafetyOUTERR2;
									
									
//Valuto la posizione in cui sta lavorando il pallettizzatore				
PortaleADx := MachinePalletizerModules.AX_X.Ax^.Status.ActPosition > 17060;//WorkSpace.X/2;		

PortaleASx := MachinePalletizerModules.AX_X.Ax^.Status.ActPosition < 17060;//WorkSpace.X/2;	

GateAccessError := MachinePalletizerGatesAccess.GateAccessConsolle.AccessERRORCode;// OR MachinePalletizerGatesAccess.GateAccess2.AccessERRORCode;
//Calcolo della formatura
_09_CalcolaFormatura();
//Calcola della lista di produzione TOTALE

IF NOT HabilitacionFormacionNueva THEN 
	_11_CalcolaListaProduzione();
ELSE
	_11_CalcolaListaProduzioneNew();	
END_IF



TimerAggancioBloccoDicurezza(IN:=I_EmergenzeOK AND PowerEnableAssi,PT:=T#2S);									
O_SbloccoFermoSicurezza := TimerAggancioBloccoDicurezza.Q;
END_ACTION

ACTION _04_Comunicazione:
AggioraDatiLgv := AggioraDatiLgv+1;
IF AggioraDatiLgv >= 250 THEN
	AggioraDatiLgv:=0;
	(* Valorizzazione della struttura dati relativa allo stato del pallettizzatore *)
	LGV_Stato_Pallettizzatore.Automatico := I_AutoPal AND MachinePalletizer_TF.IN.Mode.Auto;// AND (MachinePalletizer_TF.CmdExe.Code = CmdDO OR MachinePalletizerLGV.LGVAccesActive);// AND MachinePalletizer_TF.CmdExe.RapidStopRequest=0 AND MachinePalletizer_TF.CmdExe.PhaseStopRequest=0; 
	LGV_Stato_Pallettizzatore.Errore     := MachinePalletizer_TF.OUT.Error;
	(* Valorizzazione della struttura dati relativa allo stato delle postazioni *)	
	LGV_PostazioniPresenti := MAXAREAPRESENT;
	FOR iLgv := 1 TO MAXAREAPRESENT DO
		LGV_Stato_Postazione[iLgv].Abilitata 		:= WorkArea[iLgv].Enable;	
		LGV_Stato_Postazione[iLgv].Stato			:= WorkAreaState[iLgv].State;
		LGV_Stato_Postazione[iLgv].Tipologia 		:= WorkArea[iLgv].Typology;	
		LGV_Stato_Postazione[iLgv].AltezzaPallet 	:= LREAL_TO_REAL(WorkAreaState[iLgv].H);
		LGV_Stato_Postazione[iLgv].CodiceFalda		:= WorkAreaState[iLgv].Code;
		LGV_Stato_Postazione[iLgv].CodiceFormatura  := WorkAreaState[iLgv].F;
		LGV_Stato_Postazione[iLgv].CodiceLavorazione:= WorkAreaState[iLgv].Code;
		LGV_Stato_Postazione[iLgv].CodicePallet		:= Forming[WorkAreaState[iLgv].F].Pallet.Code;
		LGV_Stato_Postazione[iLgv].LGV_Req			:= WorkAreaState[iLgv].LGV_Req;
		LGV_Stato_Postazione[iLgv].LGVAttr			:= WorkAreaState[iLgv].LGVAttr;
		LGV_Stato_Postazione[iLgv].NPaccoSuccesivo	:= WorkAreaState[iLgv].P;
		//LGV_Stato_Postazione[iLgv].PN				:= WorkAreaState[iLgv].PN;
		LGV_Stato_Postazione[iLgv].ProgressiveNr    := TO_UDINT(WorkAreaState[iLgv].ID);
		LGV_Stato_Postazione[iLgv].Stato			:= WorkAreaState[iLgv].State;
		IF I_LGV_Stato_Operazione[iLgv] = LGV_PRELIEVO_EFFETTUATO THEN
			I_LGV_Stato_Operazione[iLgv] := LGV_OPERAZIONE_VERIFICATA;	
			I_PHPresenzaPalletVirtuale[iLgv] := FALSE;
		ELSIF I_LGV_Stato_Operazione[iLgv] = LGV_DEPOSITO_EFFETTUATO THEN
			I_LGV_Stato_Operazione[iLgv] := LGV_OPERAZIONE_VERIFICATA;	
			I_PHPresenzaPalletVirtuale[iLgv] := TRUE;
		END_IF
	END_FOR
	(* Valorizzazione della struttura dati relativa alla formatura *)
	FOR iLgv := 1 TO MAXFORMING DO
		//LGV_Stato_Formatura[iLgv].CodiceFalda := Forming[iLgv].Layer;
		//LGV_Stato_Formatura[iLgv].CodicePallet := Forming[iLgv].Pallet;
		FOR iLgvPackP := 1 TO MAXFORMINGPACK DO
			;
			//IF Forming[iLgv].PackXP[iLgvPackP].Grip <> -1 THEN
			//	LGV_Stato_Formatura[iLgv].PacchiPresenti_ZonaPositiva := UINT_TO_INT(iLgvPackP);
			//END_IF
		END_FOR
		FOR iLgvPackN := 1 TO MAXFORMINGPACK DO
			;
			//IF Forming[iLgv].PackXP[iLgvPackN].Grip <> -1 THEN
			//	LGV_Stato_Formatura[iLgv].PacchiPresenti_ZonaNegativa := UINT_TO_INT(iLgvPackN);
			//END_IF
		END_FOR
	END_FOR
	(* Gestione Richieste Ingresso *)
	(*OLGV_Req := O_LGV_Req;
	OLGV_LetIn := O_LGV_LetIn; 	
	
	ILGV_LetIn := I_LGV_LetIn;
	//ILGV_LetIn_HW := I_LGV_LetIn_HW; 		
	ILGV_LetIn_SW := I_LGV_LetIn_SW;
	ILGV_Footprint := I_LGV_Footprint;		
	//ILGV_Footprint_HW := I_LGV_Footprint_HW;	
	ILGV_Footprint_SW := I_LGV_Footprint_SW;*)
	
	////////////////////////////////////SIMULAZIONE FOTOCELLULA//////////////////////////////////////
	
	
	
	
END_IF
END_ACTION

ACTION _05_ManualCmds:
(* ******************************************************************************************************** *)
(* Machine Palletizer Modules *)
(* ******************************************************************************************************** *)
(* Robot *)
IF MachinePalletizer_TF.IN.Mode.Man AND
	(MachinePalletizer_TF.CmdExe.Code = CmdNOP OR MachinePalletizer_TF.CmdExe.Code = CmdMAN) THEN
	
	IF ManCmdGeneralHomeTRIG AND 
		MachinePalletizer_TF.Modules^.AX_X.CmdExe.Code = CmdNOP AND
		MachinePalletizer_TF.Modules^.AX_Y.CmdExe.Code = CmdNOP AND
		MachinePalletizer_TF.Modules^.AX_Z.CmdExe.Code = CmdNOP AND
		MachinePalletizer_TF.Modules^.AX_J.CmdExe.Code = CmdNOP AND
		MachinePalletizer_TF.Modules^.Pinza.CmdExe.Code = CmdNOP THEN
		ManCmdGeneralHomeTRIG := FALSE;
		MachinePalletizer_TF.ManCmd^.GeneralHome:= FALSE;
	END_IF
	IF MachinePalletizer_TF.ManCmd^.GeneralHome  AND NOT ManCmdGeneralHomeTRIG THEN
		ManCmdGeneralHomeTRIG := TRUE;
		TFParametersArrayClear(ADR(ParametersArray));
		TFCommandSend(CmdHOME,ParametersArray,MachinePalletizer_TF.Cmd);
		(*TFCommandSend(CmdHOME,ParametersArray,MachinePalletizer_TF.ModuleAX_X^.Cmd);
		TFCommandSend(CmdHOME,ParametersArray,MachinePalletizer_TF.ModuleAX_Y^.Cmd);
		TFCommandSend(CmdHOME,ParametersArray,MachinePalletizer_TF.ModuleAX_Z^.Cmd);
		TFCommandSend(CmdHOME,ParametersArray,MachinePalletizer_TF.ModuleAX_K^.Cmd);
		TFCommandSend(CmdHOME,ParametersArray,MachinePalletizer_TF.ModuleAX_J^.Cmd);
		TFCommandSend(CmdHOME,ParametersArray,MachinePalletizer_TF.ModuleAspirazione^.Cmd);*)
	END_IF
	
	(* Suction *)
	IF MachinePalletizer_TF.ManCmd^.SuctionOff THEN
		TFParametersArrayClear(ADR(ParametersArray));
		ParametersArray.Parameters[0] := '1';
		ParametersArray.Parameters[1] := '10';
		TFCommandSend(CmdMAN,ParametersArray,MachinePalletizer_TF.Modules^.Pinza.Cmd);
	ELSIF MachinePalletizer_TF.ManCmd^.SuctionOn THEN
		TFParametersArrayClear(ADR(ParametersArray));
		ParametersArray.Parameters[0] := '1';
		ParametersArray.Parameters[1] := '11';
		TFCommandSend(CmdMAN,ParametersArray,MachinePalletizer_TF.Modules^.Pinza.Cmd);
	ELSIF MachinePalletizer_TF.ManCmd^.SuctionUp THEN
		TFParametersArrayClear(ADR(ParametersArray));
		ParametersArray.Parameters[0] := '1';
		ParametersArray.Parameters[1] := '20';
		TFCommandSend(CmdMAN,ParametersArray,MachinePalletizer_TF.Modules^.Pinza.Cmd);		
	ELSIF MachinePalletizer_TF.ManCmd^.SuctionDown THEN
		TFParametersArrayClear(ADR(ParametersArray));
		ParametersArray.Parameters[0] := '1';
		ParametersArray.Parameters[1] := '21';
		TFCommandSend(CmdMAN,ParametersArray,MachinePalletizer_TF.Modules^.Pinza.Cmd);		
	END_IF

	(* X *)
	
	IF InvertiComandoJog_X THEN
		IF MachinePalletizer_TF.ManCmd^.X.JogPos THEN
			CmdJogNeg_X := TRUE;
		ELSIF MachinePalletizer_TF.ManCmd^.X.JogNeg THEN
			CmdJogPos_X := TRUE;
		END_IF
	ELSE
		IF MachinePalletizer_TF.ManCmd^.X.JogPos THEN
			CmdJogPos_X := TRUE;
		ELSIF MachinePalletizer_TF.ManCmd^.X.JogNeg THEN
			CmdJogNeg_X := TRUE;
		END_IF
	END_IF
	
	IF ManCmdXHomeTRIG AND MachinePalletizer_TF.CmdExe.Code = CmdNOP THEN
		ManCmdXHomeTRIG := FALSE;
	END_IF
	IF MachinePalletizer_TF.ManCmd^.X.Home AND NOT ManCmdXHomeTRIG THEN
		ManCmdXHomeTRIG := TRUE;
		TFParametersArrayClear(ADR(ParametersArray));
		//TFCommandSend(CmdHOME,ParametersArray,MachinePalletizer_TF.ModuleAX_X^.Cmd);
		ParametersArray.Parameters[0] := '100';
		ParametersArray.Parameters[1] := '20';
		TFCommandSend(CmdMAN,ParametersArray,MachinePalletizer_TF.Modules^.AX_X.Cmd);
	ELSIF CmdJogPos_X THEN//MachinePalletizer_TF.ManCmd^.X.JogPos THEN
		TFParametersArrayClear(ADR(ParametersArray));
		ParametersArray.Parameters[0] := '100';
		ParametersArray.Parameters[1] := '11';
		TFCommandSend(CmdMAN,ParametersArray,MachinePalletizer_TF.Modules^.AX_X.Cmd);
	ELSIF CmdJogNeg_X THEN//MachinePalletizer_TF.ManCmd^.X.JogNeg THEN
		TFParametersArrayClear(ADR(ParametersArray));
		ParametersArray.Parameters[0] := '100';
		ParametersArray.Parameters[1] := '12';
		TFCommandSend(CmdMAN,ParametersArray,MachinePalletizer_TF.Modules^.AX_X.Cmd);
	END_IF
	
	CmdJogPos_X := FALSE;
	CmdJogNeg_X := FALSE;

	(* Y *)
	IF ManCmdYHomeTRIG AND MachinePalletizer_TF.Modules^.AX_Y.CmdExe.Code = CmdNOP THEN
		ManCmdYHomeTRIG := FALSE;
	END_IF
	IF MachinePalletizer_TF.ManCmd^.Y.Home AND NOT ManCmdYHomeTRIG THEN
		ManCmdYHomeTRIG := TRUE;
		TFParametersArrayClear(ADR(ParametersArray));
		//TFCommandSend(CmdHOME,ParametersArray,MachinePalletizer_TF.ModuleAX_Y^.Cmd);
		ParametersArray.Parameters[0] := '100';
		ParametersArray.Parameters[1] := '20';
		TFCommandSend(CmdMAN,ParametersArray,MachinePalletizer_TF.Modules^.AX_Y.Cmd);
	ELSIF MachinePalletizer_TF.ManCmd^.Y.JogPos THEN
		TFParametersArrayClear(ADR(ParametersArray));
		ParametersArray.Parameters[0] := '100';
		ParametersArray.Parameters[1] := '11';
		TFCommandSend(CmdMAN,ParametersArray,MachinePalletizer_TF.Modules^.AX_Y.Cmd);
	ELSIF MachinePalletizer_TF.ManCmd^.Y.JogNeg THEN
		TFParametersArrayClear(ADR(ParametersArray));
		ParametersArray.Parameters[0] := '100';
		ParametersArray.Parameters[1] := '12';
		TFCommandSend(CmdMAN,ParametersArray,MachinePalletizer_TF.Modules^.AX_Y.Cmd);
	END_IF

	(* Z *)
	IF ManCmdZHomeTRIG AND MachinePalletizer_TF.Modules^.AX_Z.CmdExe.Code = CmdNOP THEN
		ManCmdZHomeTRIG := FALSE;
	END_IF
	IF MachinePalletizer_TF.ManCmd^.Z.Home AND NOT ManCmdZHomeTRIG THEN
		ManCmdZHomeTRIG := TRUE;
		TFParametersArrayClear(ADR(ParametersArray));
		//TFCommandSend(CmdHOME,ParametersArray,MachinePalletizer_TF.ModuleAX_Z^.Cmd);
		ParametersArray.Parameters[0] := '100';
		ParametersArray.Parameters[1] := '20';
		TFCommandSend(CmdMAN,ParametersArray,MachinePalletizer_TF.Modules^.AX_Z.Cmd);
	ELSIF MachinePalletizer_TF.ManCmd^.Z.JogPos THEN
		TFParametersArrayClear(ADR(ParametersArray));
		ParametersArray.Parameters[0] := '100';
		ParametersArray.Parameters[1] := '11';
		TFCommandSend(CmdMAN,ParametersArray,MachinePalletizer_TF.Modules^.AX_Z.Cmd);
	ELSIF MachinePalletizer_TF.ManCmd^.Z.JogNeg THEN
		TFParametersArrayClear(ADR(ParametersArray));
		ParametersArray.Parameters[0] := '100';
		ParametersArray.Parameters[1] := '12';
		TFCommandSend(CmdMAN,ParametersArray,MachinePalletizer_TF.Modules^.AX_Z.Cmd);
	END_IF

	(* J *)
	IF ManCmdJHomeTRIG AND MachinePalletizer_TF.Modules^.AX_J.CmdExe.Code = CmdNOP THEN
		ManCmdJHomeTRIG := FALSE;
	END_IF
	IF MachinePalletizer_TF.ManCmd^.J.Home AND NOT ManCmdJHomeTRIG THEN
		ManCmdJHomeTRIG := TRUE;
		TFParametersArrayClear(ADR(ParametersArray));
		//TFCommandSend(CmdHOME,ParametersArray,MachinePalletizer_TF.ModuleAX_J^.Cmd);
		ParametersArray.Parameters[0] := '100';
		ParametersArray.Parameters[1] := '20';
		TFCommandSend(CmdMAN,ParametersArray,MachinePalletizer_TF.Modules^.AX_J.Cmd);
	ELSIF MachinePalletizer_TF.ManCmd^.J.JogPos THEN
		TFParametersArrayClear(ADR(ParametersArray));
		ParametersArray.Parameters[0] := '100';
		ParametersArray.Parameters[1] := '11';
		TFCommandSend(CmdMAN,ParametersArray,MachinePalletizer_TF.Modules^.AX_J.Cmd);
	ELSIF MachinePalletizer_TF.ManCmd^.J.JogNeg THEN
		TFParametersArrayClear(ADR(ParametersArray));
		ParametersArray.Parameters[0] := '100';
		ParametersArray.Parameters[1] := '12';
		TFCommandSend(CmdMAN,ParametersArray,MachinePalletizer_TF.Modules^.AX_J.Cmd);
	END_IF

	(* PINZA: ASPIRAZIONE/APERTURA CHIUSURA *)
	IF ManCmdJHomeTRIG AND MachinePalletizer_TF.Modules^.AX_J.CmdExe.Code = CmdNOP THEN
		ManCmdJHomeTRIG := FALSE;
	END_IF
	IF MachinePalletizer_TF.ManCmd^.Pinza.ApriPinza THEN
		TFParametersArrayClear(ADR(ParametersArray));
		ParametersArray.Parameters[0] := '1';
		ParametersArray.Parameters[1] := '10';
		TFCommandSend(CmdMAN,ParametersArray,MachinePalletizer_TF.Modules^.Pinza.Cmd);
		MachinePalletizer_TF.ManCmd^.Pinza.ApriPinza := FALSE;
	END_IF
	IF MachinePalletizer_TF.ManCmd^.Pinza.ChiudiPinza THEN
		TFParametersArrayClear(ADR(ParametersArray));
		ParametersArray.Parameters[0] := '1';
		ParametersArray.Parameters[1] := '11';
		MachinePalletizer_TF.ManCmd^.Pinza.ChiudiPinza := FALSE;
		TFCommandSend(CmdMAN,ParametersArray,MachinePalletizer_TF.Modules^.Pinza.Cmd);
	END_IF
	IF MachinePalletizer_TF.ManCmd^.Pinza.SbloccoPinza THEN
		TFParametersArrayClear(ADR(ParametersArray));
		ParametersArray.Parameters[0] := '1';
		ParametersArray.Parameters[1] := '20';
		MachinePalletizer_TF.ManCmd^.Pinza.SbloccoPinza:= FALSE;
		TFCommandSend(CmdMAN,ParametersArray,MachinePalletizer_TF.Modules^.Pinza.Cmd);
	END_IF
	IF MachinePalletizer_TF.ManCmd^.Pinza.BloccoPinza THEN
		TFParametersArrayClear(ADR(ParametersArray));
		ParametersArray.Parameters[0] := '1';
		ParametersArray.Parameters[1] := '21';
		MachinePalletizer_TF.ManCmd^.Pinza.BloccoPinza:= FALSE;
		TFCommandSend(CmdMAN,ParametersArray,MachinePalletizer_TF.Modules^.Pinza.Cmd);
	END_IF
	IF MachinePalletizer_TF.ManCmd^.Pinza.AttivazioneVuotoFaldeDX THEN
		TFParametersArrayClear(ADR(ParametersArray));
		ParametersArray.Parameters[0] := '1';
		ParametersArray.Parameters[1] := '30';
		MachinePalletizer_TF.ManCmd^.Pinza.AttivazioneVuotoFaldeDX := FALSE;
		TFCommandSend(CmdMAN,ParametersArray,MachinePalletizer_TF.Modules^.Pinza.Cmd);
	END_IF
	IF MachinePalletizer_TF.ManCmd^.Pinza.DisattivazioneVuotoFaldeDX THEN
		TFParametersArrayClear(ADR(ParametersArray));
		ParametersArray.Parameters[0] := '1';
		ParametersArray.Parameters[1] := '31';
		MachinePalletizer_TF.ManCmd^.Pinza.DisattivazioneVuotoFaldeDX := FALSE;
		TFCommandSend(CmdMAN,ParametersArray,MachinePalletizer_TF.Modules^.Pinza.Cmd);
	END_IF
	IF MachinePalletizer_TF.ManCmd^.Pinza.AttivazioneVuotoFaldeSX THEN
		TFParametersArrayClear(ADR(ParametersArray));
		ParametersArray.Parameters[0] := '1';
		ParametersArray.Parameters[1] := '40';
		MachinePalletizer_TF.ManCmd^.Pinza.AttivazioneVuotoFaldeSX := FALSE;
		TFCommandSend(CmdMAN,ParametersArray,MachinePalletizer_TF.Modules^.Pinza.Cmd);
	END_IF
	IF MachinePalletizer_TF.ManCmd^.Pinza.DisattivazioneVuotoFaldeSX THEN
		TFParametersArrayClear(ADR(ParametersArray));
		ParametersArray.Parameters[0] := '1';
		ParametersArray.Parameters[1] := '41';
		MachinePalletizer_TF.ManCmd^.Pinza.DisattivazioneVuotoFaldeSX := FALSE;
		TFCommandSend(CmdMAN,ParametersArray,MachinePalletizer_TF.Modules^.Pinza.Cmd);
	END_IF
	IF MachinePalletizer_TF.ManCmd^.Pinza.AttivazioneVuotoDX THEN
		TFParametersArrayClear(ADR(ParametersArray));
		ParametersArray.Parameters[0] := '1';
		ParametersArray.Parameters[1] := '50';
		MachinePalletizer_TF.ManCmd^.Pinza.AttivazioneVuotoDX := FALSE;
		TFCommandSend(CmdMAN,ParametersArray,MachinePalletizer_TF.Modules^.Pinza.Cmd);
	END_IF
//	IF MachinePalletizer_TF.ManCmd^.Pinza.DisattivazioneVuotoDX THEN
//		TFParametersArrayClear(ADR(ParametersArray));
//		ParametersArray.Parameters[0] := '1';
//		ParametersArray.Parameters[1] := '51';
//		MachinePalletizer_TF.ManCmd^.Pinza.DisattivazioneVuotoDX := FALSE;
//		TFCommandSend(CmdMAN,ParametersArray,MachinePalletizer_TF.Modules^.Pinza.Cmd);
//	END_IF
	IF MachinePalletizer_TF.ManCmd^.Pinza.AttivazioneVuotoSX THEN
		TFParametersArrayClear(ADR(ParametersArray));
		ParametersArray.Parameters[0] := '1';
		ParametersArray.Parameters[1] := '60';
		MachinePalletizer_TF.ManCmd^.Pinza.AttivazioneVuotoSX := FALSE;
		TFCommandSend(CmdMAN,ParametersArray,MachinePalletizer_TF.Modules^.Pinza.Cmd);
	END_IF
	IF MachinePalletizer_TF.ManCmd^.Pinza.DisattivazioneVuotoSX THEN
		
		IF Ciclo_Deposito_Lastra.Stato <> ANNULLATO AND NOT EseguitoAllinementoPezziDeposito(*AND MachinePalletizer_TF.Modules^.Pinza.AspirazioneSX^.Out.Attiva_Vuoto AND MachinePalletizer_TF.Modules^.Pinza.StatoPinza.LatoSxPiastrellaInPresa*) THEN
			IF Mission.PPlace > 0 THEN
				//Aggiungo la lastra in deposito e aggiorno lo stato della lastra della lista in modo da contrasegnarla elaborata 
				IF (MachinePalletizerModules.AX_X.Ax^.AxRef^.NcToPlc.ActPos >= WorkArea[Mission.PPlace].X - 300) AND 
					(MachinePalletizerModules.AX_X.Ax^.AxRef^.NcToPlc.ActPos <= WorkArea[Mission.PPlace].X + 300) THEN
					//WorkAreaState[Mission.PPlace].Slab[WorkAreaState[Mission.PPlace].P] 	:= MachinePalletizerModules.Pinza.ElementoInPrelievo^;
					//WorkAreaState[Mission.PPlace].SlabData[WorkAreaState[Mission.PPlace].P] := MachinePalletizerModules.Pinza.DataElement^;
					WorkAreaState[Mission.PPlace].P := WorkAreaState[Mission.PPlace].P +1;
					HMI_NumeroPezziPresentiPostazione[Mission.PPlace] := HMI_NumeroPezziPresentiPostazione[Mission.PPlace] + 1;
					IF  WorkAreaState[Mission.PPlace].Supporto.Tipologia = CAVALLETTO  THEN
						IF PosicionJDestino = 0 THEN
							WorkAreaState[Mission.PPlace].P_Cava.HMI_NumeroPezziPresentiPostazione_A_Cavaleto := WorkAreaState[Mission.PPlace].P_Cava.HMI_NumeroPezziPresentiPostazione_A_Cavaleto+1;
							HMI_NumeroPezziPresentiCavallete[Mission.PPlace].HMI_NumeroPezziPresentiPostazione_A_Cavaleto := HMI_NumeroPezziPresentiCavallete[Mission.PPlace].HMI_NumeroPezziPresentiPostazione_A_Cavaleto +1 ;
						END_IF
						IF PosicionJDestino = 180 THEN
							WorkAreaState[Mission.PPlace].P_Cava.HMI_NumeroPezziPresentiPostazione_B_Cavaleto := WorkAreaState[Mission.PPlace].P_Cava.HMI_NumeroPezziPresentiPostazione_B_Cavaleto+1;
							HMI_NumeroPezziPresentiCavallete[Mission.PPlace].HMI_NumeroPezziPresentiPostazione_B_Cavaleto := HMI_NumeroPezziPresentiCavallete[Mission.PPlace].HMI_NumeroPezziPresentiPostazione_B_Cavaleto +1 ;
						END_IF 
					END_IF
					
					FOR i := 1 TO MAXELEMENTLIST DO
						IF WorkAreaProductionList[Mission.PPlace].PElementList[i].Stato = ELEMENTO_DA_ELABORARE THEN
							WorkAreaProductionList[Mission.PPlace].PElementList[i].Stato := ELEMENTO_ELABORATO; //Dichiaro che l'elemento della lista è stato elaborato
							EXIT;
						END_IF
					END_FOR	
					EseguitoAllinementoPezziDeposito := TRUE;				
				ELSE
					;
				END_IF
				//aggiungo nel prelievo la lastra se è stata rimessa al suo posto
				IF (MachinePalletizerModules.AX_X.Ax^.AxRef^.NcToPlc.ActPos >= WorkArea[Mission.PPick].X - 300) AND 
					(MachinePalletizerModules.AX_X.Ax^.AxRef^.NcToPlc.ActPos <= WorkArea[Mission.PPick].X + 300) THEN
					//WorkAreaState[Mission.PPlace].Slab[WorkAreaState[Mission.PPlace].P] 	:= MachinePalletizerModules.Pinza.ElementoInPrelievo^;
					//WorkAreaState[Mission.PPlace].SlabData[WorkAreaState[Mission.PPlace].P] := MachinePalletizerModules.Pinza.DataElement^;
					WorkAreaState[Mission.PPick].P := WorkAreaState[Mission.PPick].P +1;
					HMI_NumeroPezziPresentiPostazione[Mission.PPick] := HMI_NumeroPezziPresentiPostazione[Mission.PPick] + 1;
					IF  WorkAreaState[Mission.PPlace].Supporto.Tipologia = CAVALLETTO  THEN
						IF PosicionJDestino = 0 THEN
							WorkAreaState[Mission.PPick].P_Cava.HMI_NumeroPezziPresentiPostazione_A_Cavaleto := WorkAreaState[Mission.PPick].P_Cava.HMI_NumeroPezziPresentiPostazione_A_Cavaleto+1;
							HMI_NumeroPezziPresentiCavallete[Mission.PPick].HMI_NumeroPezziPresentiPostazione_A_Cavaleto := HMI_NumeroPezziPresentiCavallete[Mission.PPick].HMI_NumeroPezziPresentiPostazione_A_Cavaleto +1 ;
						END_IF
						IF PosicionJDestino = 180 THEN
							WorkAreaState[Mission.PPick].P_Cava.HMI_NumeroPezziPresentiPostazione_B_Cavaleto := WorkAreaState[Mission.PPick].P_Cava.HMI_NumeroPezziPresentiPostazione_B_Cavaleto+1;
							HMI_NumeroPezziPresentiCavallete[Mission.PPick].HMI_NumeroPezziPresentiPostazione_B_Cavaleto := HMI_NumeroPezziPresentiCavallete[Mission.PPick].HMI_NumeroPezziPresentiPostazione_B_Cavaleto +1 ;
						END_IF 
					END_IF
					EseguitoAllinementoPezziDeposito := TRUE;	
				ELSE
					;
				END_IF
			END_IF
			
		END_IF
	
		TFParametersArrayClear(ADR(ParametersArray));
		ParametersArray.Parameters[0] := '1';
		ParametersArray.Parameters[1] := '61';
		MachinePalletizer_TF.ManCmd^.Pinza.DisattivazioneVuotoSX := FALSE;
		TFCommandSend(CmdMAN,ParametersArray,MachinePalletizer_TF.Modules^.Pinza.Cmd);
		Ciclo_Prelievo_Lastra.Stato 		:= ANNULLATO;
		Ciclo_Pelievo_Falda.Stato 			:= ANNULLATO;
		Ciclo_Deposito_Lastra.Stato			:= ANNULLATO;
		Ciclo_Deposito_Falda.Stato			:= ANNULLATO;
		Ciclo_Di_Riposo.Stato				:= ANNULLATO;
		Ciclo_Prelievo_Lastra_Depal.Stato 	:= ANNULLATO;
		Ciclo_Deposito_Lastra_Depal.Stato 	:= ANNULLATO;
		Ciclo_Deposito_Falda_Depal.Stato 	:= ANNULLATO;
		ProductOnGripper 					:= KNOPRODUCT;
		Ciclo_Deposito_Falda_Depal.Stato 	:= ANNULLATO;
		
		//Azzero hli apprendimenti e riporto le quote allo stato iniziale
		FOR i:=1 TO MAXAREAPRESENT DO
			WorkAreaState[i].Apprendimento.Z.Lato0.Stato 	:= APPRENDIMENTO_DA_ESEGUIRE;
			WorkAreaState[i].Apprendimento.Z.Lato90.Stato 	:= APPRENDIMENTO_DA_ESEGUIRE;
			WorkAreaState[i].Apprendimento.Z.Lato180.Stato 	:= APPRENDIMENTO_DA_ESEGUIRE;
		END_FOR
		
		StatoMissione 				:= MISSION_STATE_NOP;//Azzero segnalazione a HMI
		WorkAreaManager.State 		:= WAMANAGER_NOP;
		Mission.State 				:= MISSION_STATE_NOP;
		MaterialeDepositatoSuLinea 	:= TRUE;//In questo modo se scarico la mattonella sulla rulliera, lei parte
	END_IF
	IF MachinePalletizer_TF.ManCmd^.Pinza.AttivaTastatori THEN
		TFParametersArrayClear(ADR(ParametersArray));
		ParametersArray.Parameters[0] := '1';
		ParametersArray.Parameters[1] := '70';
		MachinePalletizer_TF.ManCmd^.Pinza.AttivaTastatori := FALSE;
		TFCommandSend(CmdMAN,ParametersArray,MachinePalletizer_TF.Modules^.Pinza.Cmd);
	END_IF
	IF MachinePalletizer_TF.ManCmd^.Pinza.DisattivaTastatori THEN
		TFParametersArrayClear(ADR(ParametersArray));
		ParametersArray.Parameters[0] := '1';
		ParametersArray.Parameters[1] := '71';
		MachinePalletizer_TF.ManCmd^.Pinza.DisattivaTastatori := FALSE;
		TFCommandSend(CmdMAN,ParametersArray,MachinePalletizer_TF.Modules^.Pinza.Cmd);
	END_IF
	IF MachinePalletizer_TF.ManCmd^.Pinza.CalibrazioneOVEM THEN
		TFParametersArrayClear(ADR(ParametersArray));
		MachinePalletizer_TF.ManCmd^.Pinza.CalibrazioneOVEM := FALSE;
		TFCommandSend(CmdHOME,ParametersArray,MachinePalletizer_TF.Modules^.Pinza.Cmd);
	END_IF

	//Posizionamento diretto pinza
	IF MachinePalletizer_TF.ManCmd^.PosizionamentoPinza0 THEN
		TFParametersArrayClear(ADR(ParametersArray));
		ParametersArray.Parameters[0] := '100';
		ParametersArray.Parameters[1] := '13';
		MachinePalletizer_TF.Modules^.AX_J.AxisPar^.Quota_Destinazione := 0;
		TFCommandSend(CmdMAN,ParametersArray,MachinePalletizer_TF.Modules^.AX_J.Cmd);
		MachinePalletizer_TF.ManCmd^.PosizionamentoPinza0 := FALSE;
	END_IF
	IF MachinePalletizer_TF.ManCmd^.PosizionamentoPinza90 THEN
		TFParametersArrayClear(ADR(ParametersArray));
		ParametersArray.Parameters[0] := '100';
		ParametersArray.Parameters[1] := '13';
		MachinePalletizer_TF.Modules^.AX_J.AxisPar^.Quota_Destinazione := 90;
		TFCommandSend(CmdMAN,ParametersArray,MachinePalletizer_TF.Modules^.AX_J.Cmd);
		 MachinePalletizer_TF.ManCmd^.PosizionamentoPinza90 := FALSE;
	END_IF
	IF MachinePalletizer_TF.ManCmd^.PosizionamentoPinza180 THEN
		TFParametersArrayClear(ADR(ParametersArray));
		ParametersArray.Parameters[0] := '100';
		ParametersArray.Parameters[1] := '13';
		MachinePalletizer_TF.Modules^.AX_J.AxisPar^.Quota_Destinazione := 180;
		TFCommandSend(CmdMAN,ParametersArray,MachinePalletizer_TF.Modules^.AX_J.Cmd);
		MachinePalletizer_TF.ManCmd^.PosizionamentoPinza180 := FALSE;
	END_IF
	
	IF ManCmdXHomeTRIG AND 
		MachinePalletizer_TF.Modules^.AX_X.CmdExe.Code = CmdNOP THEN
		ManCmdXHomeTRIG := FALSE;
		MachinePalletizer_TF.ManCmd^.X.Home:= FALSE;
	END_IF
	IF ManCmdYHomeTRIG AND 
		MachinePalletizer_TF.Modules^.AX_Y.CmdExe.Code = CmdNOP THEN
		ManCmdYHomeTRIG := FALSE;
		MachinePalletizer_TF.ManCmd^.Y.Home:= FALSE;
	END_IF
	IF ManCmdZHomeTRIG AND 
		MachinePalletizer_TF.Modules^.AX_Z.CmdExe.Code = CmdNOP THEN
		ManCmdZHomeTRIG := FALSE;
		MachinePalletizer_TF.ManCmd^.Z.Home:= FALSE;
	END_IF
	IF ManCmdJHomeTRIG AND 
		MachinePalletizer_TF.Modules^.AX_J.CmdExe.Code = CmdNOP THEN
		ManCmdJHomeTRIG := FALSE;
		MachinePalletizer_TF.ManCmd^.J.Home:= FALSE;
	END_IF
	
END_IF
END_ACTION

ACTION _06_ScriviOutput:
(* Control Word OVEM *)
O_ControlWordOVEM_1 := MachinePalletizerModules.Pinza.AspirazioneDX1^.Out.ControlWord;
O_ControlWordOVEM_2 := MachinePalletizerModules.Pinza.AspirazioneSX1^.Out.ControlWord;

O_ControlWordOVEM_12 := MachinePalletizerModules.Pinza.AspirazioneDX2^.Out.ControlWord;
O_ControlWordOVEM_22 := MachinePalletizerModules.Pinza.AspirazioneSX2^.Out.ControlWord;

(* Configurazione Porte Ciabatta Pinza *)

{info 'TODO:SISTEMARE IO PINZA'}	

//Q_K517[22] := 1; //Configurazione pin 2 e pin 4 come uscite porta X1.0
//Q_K517[23] := 1; //Configurazione pin 2 e pin 4 come uscite porta X1.1
//Q_K517[24] := 1; //Configurazione pin 2 e pin 4 come uscite porta X1.2
Q_K517[25] := 1; //Configurazione pin 2 e pin 4 come uscite porta X1.3
//Q_K517[26] := 1; //Configurazione pin 2 e pin 4 come uscite porta X1.4
//Q_K517[27] := 1; //Configurazione pin 2 e pin 4 come uscite porta X1.5
Q_K517[28] := 1; //Configurazione pin 2 e pin 4 come uscite porta X1.6
Q_K517[29] := 1; //Configurazione pin 2 e pin 4 come uscite porta X1.7

//Q_K517[2].0 //Comando X1.0 pin 4
//Q_K517[2].1 //Comando X1.1 pin 4
//Q_K517[2].2 //Comando X1.2 pin 4
//Q_K517[2].3 //Comando X1.3 pin 4
//Q_K517[2].4 //Comando X1.4 pin 4
//Q_K517[2].5 //Comando X1.5 pin 4
//Q_K517[2].6 //Comando X1.6 pin 4
//Q_K517[2].7 //Comando X1.7 pin 4
///------------------------------//
//Q_K517[3].0 //Comando X1.0 pin 2
//Q_K517[3].1 //Comando X1.1 pin 2
//Q_K517[3].2 //Comando X1.2 pin 2
//Q_K517[3].3 //Comando X1.3 pin 2
//Q_K517[3].4 //Comando X1.4 pin 2
//Q_K517[3].5 //Comando X1.5 pin 2
//Q_K517[3].6 //Comando X1.6 pin 2
//Q_K517[3].7 //Comando X1.7 pin 2

Q_K517[2].3 := MachinePalletizerModules.Pinza.AspirazioneFaldaDX^.OUT.ActivationOutput;
Q_K517[2].6 := MachinePalletizerModules.Pinza.CilindroSbloccoBascolante^.OUT.ActivationOutput;
Q_K517[2].7 := MachinePalletizerModules.Pinza.CilindroSbloccoRotazione^.OUT.ActivationOutput;

//Q_J17[3].7 := MachinePalletizerModules.Pinza.CilindroTasteggio^.OUT.ActivationOutput;

LetturaFTCPinza0_1 		:= MachinePalletizerModules.Pinza.StatoPinza.LetturaFTC0;
LetturaFTCPinza180_1 	:= MachinePalletizerModules.Pinza.StatoPinza.LetturaFTC180;
LetturaFTCPinza0_2 		:= MachinePalletizerModules.Pinza.StatoPinza.LetturaFTC0_2;
LetturaFTCPinza180_2 	:= MachinePalletizerModules.Pinza.StatoPinza.LetturaFTC180_2;

(* ******************************************************************************************************** *)
(* OUTPUT Transfer *)
(* ******************************************************************************************************** *)

(* Pallet and Layer stacks state *)
PalletStackEmpty 												:= MachinePalletizer_TF.PalletStackEmpty;
LayerStackEmpty 												:= MachinePalletizer_TF.LayerStackEmpty;
AllWABusy 														:= MachinePalletizer_TF.AllWABusy;

(* Machine Palletizer *)
O_ResetACKAzionamenti 	:= I_StartCicloPal OR MachinePalletizerGatesAccess.GateAccessConsolle.ErrAckDriver;// OR MachinePalletizerGatesAccess.GateAccess2.ErrAckDriver;// OR MachinePalletizerLGV.ErrAckDriver;
O_AbilitazioneMarcia	:= MachinePalletizer_TF.OUT.PowerActive;


O_SirenaAllarmiPal		:= MachinePalletizer_TF.OUT.StartHorn OR MachinePalletizer_TF.OUT.Horn OR (MachinePalletizer_TF.OUT.Warning AND MachinePalletizer_TF.OUT.ClockSegnalazioniAlternato AND NOT MachinePalletizer_TF.OUT.ResetSirenaSegnalazioni);// OR (I_Trasporti_GEN_GLOBAL_ALARM_STOP AND MachinePalletizer_TF.OUT.ClockSegnalazioni);

O_LampadaAutomaticoPal	:= MachinePalletizer_TF.OUT.Run;

O_LampadaAllarmiPal		:= (MachinePalletizer_TF.OUT.Error AND MachinePalletizer_TF.OUT.ClockSegnalazioni) OR
							MachinePalletizer_TF.OUT.Error;
							
																	
O_Reset_Plc_Sicurezza := I_StartCicloPal OR 
						MachinePalletizerGatesAccess.GateAccessConsolle.ErrAck OR
						MachinePalletizerGatesAccess.GateAccessPS306.ErrAck OR
						MachinePalletizerGatesAccess.GateAccessPS307.ErrAck OR
						MachinePalletizerGatesAccess.GateAccessPS308.ErrAck OR
						MachinePalletizerGatesAccess.GateAccessPS309.ErrAck;


O_LampadaPulsanteCicloPalConsolle:= MachinePalletizer_TF.OUT.Run OR 
									(ResetNecessarioCentralinaSafety AND MachinePalletizer_TF.OUT.ClockSegnalazioni) ;
O_LampadaPulsanteMarciaPalConsolle := I_MarciaOK AND (MachinePalletizerModules.AX_X.Ax^.Status.PowerActive AND 
													MachinePalletizerModules.AX_Y.Ax^.Status.PowerActive AND 
													MachinePalletizerModules.AX_Z.Ax^.Status.PowerActive AND 
													MachinePalletizerModules.AX_J.Ax^.Status.PowerActive) OR 
										((I_MarciaOK AND NOT(MachinePalletizerModules.AX_X.Ax^.Status.PowerActive AND 
														MachinePalletizerModules.AX_Y.Ax^.Status.PowerActive AND 
														MachinePalletizerModules.AX_Z.Ax^.Status.PowerActive AND 
														MachinePalletizerModules.AX_J.Ax^.Status.PowerActive) OR
										(I_SafetyStateEmergenze_Generali <> 1 OR 
                                          I_SafetyStateEmergenza_PS306_307 <> 1 OR
                                          I_SafetyStateEmergenza_PS308_309 <> 1)) AND MachinePalletizer_TF.OUT.ClockSegnalazioni)AND NOT ResetNecessarioCentralinaSafety;

(* Gates Access *)
O_LampadaRichiestaIngressoPal	:= (MachinePalletizerGatesAccess.GateAccessConsolle.AccessLamp OR 
									MachinePalletizerGatesAccess.GateAccessPS306.AccessLamp OR
									MachinePalletizerGatesAccess.GateAccessPS307.AccessLamp OR 
									MachinePalletizerGatesAccess.GateAccessPS308.AccessLamp OR 
									MachinePalletizerGatesAccess.GateAccessPS309.AccessLamp OR
									(NOT I_BarrierePallettizzatoreOK AND MachinePalletizer_TF.OUT.ClockSegnalazioni))AND NOT ResetNecessarioCentralinaSafety;

O_LampadaPulsanteRichiestaIngressoConsolle := MachinePalletizerGatesAccess.GateAccessConsolle.AccessLamp OR 
											((I_BarrierePallettizzatoreOK <> 1 AND MachinePalletizer_TF.OUT.ClockSegnalazioni) AND NOT ResetNecessarioCentralinaSafety);
									
O_LampadaPulsanteRichiestaIngressoPS306 := MachinePalletizerGatesAccess.GateAccessPS306.AccessLamp OR 
											((NOT I_BarrierePallettizzatoreOK AND MachinePalletizer_TF.OUT.ClockSegnalazioni) AND NOT ResetNecessarioCentralinaSafety);

O_LampadaPulsanteRichiestaIngressoPS307 := MachinePalletizerGatesAccess.GateAccessPS307.AccessLamp OR 
											((NOT I_BarrierePallettizzatoreOK AND MachinePalletizer_TF.OUT.ClockSegnalazioni) AND NOT ResetNecessarioCentralinaSafety);

O_LampadaPulsanteRichiestaIngressoPS308 := MachinePalletizerGatesAccess.GateAccessPS308.AccessLamp OR 
											((NOT I_BarrierePallettizzatoreOK AND MachinePalletizer_TF.OUT.ClockSegnalazioni) AND NOT ResetNecessarioCentralinaSafety);

O_LampadaPulsanteRichiestaIngressoPS309 := MachinePalletizerGatesAccess.GateAccessPS309.AccessLamp OR 
											((NOT I_BarrierePallettizzatoreOK AND MachinePalletizer_TF.OUT.ClockSegnalazioni) AND NOT ResetNecessarioCentralinaSafety);
									
//******************** SCHEDA OUT AP201.4
O_AP201_4[1]	:= O_SirenaAllarmiPal;				
O_AP201_4[2]	:= O_LampadaAutomaticoPal;			
O_AP201_4[3]	:= O_LampadaAllarmiPal;				
O_AP201_4[4]	:= O_LampadaRichiestaIngressoPal;
O_AP201_4[5]	:= O_ConsensoVeicolo[1];						
O_AP201_4[6]	:= O_ConsensoVeicolo[2];						
O_AP201_4[7]	:= O_ConsensoVeicolo[3];						
O_AP201_4[8]	:= O_ConsensoVeicolo[4];						
O_AP201_4[9]	:= O_LampadaPulsanteCicloPalConsolle; 			
O_AP201_4[10]	:= O_LampadaPulsanteRichiestaIngressoConsolle; 	
O_AP201_4[11]	:= O_LampadaPulsanteMarciaPalConsolle;			
O_AP201_4[12]	:= O_LampadaPulsanteRichiestaIngressoPS306; 	
O_AP201_4[13]	:= O_LampadaPulsanteRichiestaIngressoPS307;		
O_AP201_4[14]	:= O_LampadaPulsanteRichiestaIngressoPS308; 	
O_AP201_4[15]	:= O_LampadaPulsanteRichiestaIngressoPS309;		
O_AP201_4[16]	:= FALSE; 										
											
//******************** SCHEDA OUT SAFETY AP201.5											
O_AP201_5;											
//O_MarciaPal	: BOOL; // CH1=											
//FREE			: BOOL; // CH2=												
//FREE			: BOOL; // CH3=												
//FREE			: BOOL; // CH4=			
									
//******************** SCHEDA OUT AP201.6												
O_AP201_6[1]	:= O_LampadaIngressoVietatoPS306; 												
O_AP201_6[2]	:= O_LampadaIngressoVietatoPS307; 												
O_AP201_6[3]	:= O_LampadaIngressoVietatoPS308; 												
O_AP201_6[4]	:= O_LampadaIngressoVietatoPS309; 												
O_AP201_6[5]	:= O_ConsensoVeicolo[5];		  												
O_AP201_6[6]	:= O_ConsensoVeicolo[6];														
O_AP201_6[7]	:= O_ConsensoVeicolo[7];														
O_AP201_6[8]	:= O_ConsensoVeicolo[8];														
O_AP201_6[9]	:= FALSE; 																		
O_AP201_6[10]	:= FALSE; 																		
O_AP201_6[11]	:= FALSE; 																		
O_AP201_6[12]	:= FALSE; 																		
O_AP201_6[13]	:= FALSE; 																		
O_AP201_6[14]	:= FALSE; 							
O_AP201_6[15]	:= FALSE; 							
O_AP201_6[16]	:= FALSE; 							


O_XDriveDigitalOutput.1 := O_SbloccoFermoSicurezza; //Sblocco del paracadute -> ingresso 1 del drive X
END_ACTION

ACTION _07_ScriviStatus:
(*Valorizzazione della struttura Status_TF*)

(*Stato Macchina*)
Status_TF.Macchina.Auto					:= MachinePalletizer_TF.IN.Mode.Auto AND MachinePalletizer_TF.CmdExe.Code = CmdDO;
Status_TF.Macchina.Run					:= MachinePalletizer_TF.OUT.Run;
Status_TF.Macchina.Error				:= MachinePalletizer_TF.Error.Code;
Status_TF.Macchina.ErrorExtra			:= MachinePalletizer_TF.Error.ExtraCode;
Status_TF.Macchina.PowerOK				:= MachinePalletizer_TF.IN.PowerOk;
Status_TF.Macchina.EmergencyOK			:= MachinePalletizer_TF.IN.Mode.EmergencyRequest;

(*Stato assi*)	
Status_TF.X.Position 					:= MachinePalletizerModules.AX_X.Ax^.Status.ActPosition;
Status_TF.X.Velocity 					:= MachinePalletizerModules.AX_X.Ax^.Status.ActVelocity;
Status_TF.X.Torque 						:= MachinePalletizerModules.AX_X.Ax^.Status.ActTorque;
Status_TF.X.Error 						:= MachinePalletizerModules.AX_X.Ax^.Status.ErrorID;
Status_TF.X.PowerActive					:= MachinePalletizerModules.AX_X.Ax^.Status.PowerActive;

Status_TF.Y.Position 					:= MachinePalletizerModules.AX_Y.Ax^.Status.ActPosition;
Status_TF.Y.Velocity 					:= MachinePalletizerModules.AX_Y.Ax^.Status.ActVelocity;
Status_TF.Y.Torque 						:= MachinePalletizerModules.AX_Y.Ax^.Status.ActTorque;
Status_TF.Y.Error 						:= MachinePalletizerModules.AX_Y.Ax^.Status.ErrorID;
Status_TF.Y.PowerActive					:= MachinePalletizerModules.AX_Y.Ax^.Status.PowerActive;

Status_TF.Z.Position 					:= MachinePalletizerModules.AX_Z.Ax^.Status.ActPosition;
Status_TF.Z.Velocity 					:= MachinePalletizerModules.AX_Z.Ax^.Status.ActVelocity;
Status_TF.Z.Torque 						:= MachinePalletizerModules.AX_Z.Ax^.Status.ActTorque;
Status_TF.Z.Error 						:= MachinePalletizerModules.AX_Z.Ax^.Status.ErrorID;
Status_TF.Z.PowerActive					:= MachinePalletizerModules.AX_Z.Ax^.Status.PowerActive;

Status_TF.J.Position 					:= MachinePalletizerModules.AX_J.Ax^.Status.ActPosition;
Status_TF.J.Velocity 					:= MachinePalletizerModules.AX_J.Ax^.Status.ActVelocity;
Status_TF.J.Torque 						:= MachinePalletizerModules.AX_J.Ax^.Status.ActTorque;
Status_TF.J.Error 						:= MachinePalletizerModules.AX_J.Ax^.Status.ErrorID;
Status_TF.J.PowerActive					:= MachinePalletizerModules.AX_J.Ax^.Status.PowerActive;

Status_TF.K.Position 					:= 0;//ModuloAsse_K.Ax^.Status.ActPosition;
Status_TF.K.Velocity 					:= 0;//ModuloAsse_K.Ax^.Status.ActVelocity;
Status_TF.K.Torque 						:= 0;//ModuloAsse_K.Ax^.Status.ActTorque;
Status_TF.K.Error 						:= 0;//ModuloAsse_K.Ax^.Status.ErrorID;
Status_TF.K.PowerActive					:= 0;//ModuloAsse_K.Ax^.Status.PowerActive;

(*Stato Moduli*)
//Status_TF.ModAsse_X.Cmd					:= ModuloAsse_X.CmdExe.Code;
//Status_TF.ModAsse_X.CmdCase				:= ModuloAsse_X.CmdExe.CmdCase;
Status_TF.ModAsse_X.Error       		:= MachinePalletizerModules.AX_X.Error.Code;
Status_TF.ModAsse_X.ErrorExtra      	:= MachinePalletizerModules.AX_X.Error.ExtraCode;

//Status_TF.ModAsse_Y.Cmd					:= ModuloAsse_Y.CmdExe.Code;
//Status_TF.ModAsse_Y.CmdCase				:= ModuloAsse_Y.CmdExe.CmdCase;
Status_TF.ModAsse_Y.Error       		:= MachinePalletizerModules.AX_Y.Error.Code;
Status_TF.ModAsse_Y.ErrorExtra      	:= MachinePalletizerModules.AX_Y.Error.ExtraCode;

//Status_TF.ModAsse_Z.Cmd					:= ModuloAsse_Z.CmdExe.Code;
//Status_TF.ModAsse_Z.CmdCase				:= ModuloAsse_Z.CmdExe.CmdCase;
Status_TF.ModAsse_Z.Error       		:= MachinePalletizerModules.AX_Z.Error.Code;
Status_TF.ModAsse_Z.ErrorExtra      	:= MachinePalletizerModules.AX_Z.Error.ExtraCode;

//Status_TF.ModAsse_J.Cmd					:= ModuloAsse_J.CmdExe.Code;
//Status_TF.ModAsse_J.CmdCase				:= ModuloAsse_J.CmdExe.CmdCase;
Status_TF.ModAsse_J.Error       		:= MachinePalletizerModules.AX_J.Error.Code;
Status_TF.ModAsse_J.ErrorExtra      	:= MachinePalletizerModules.AX_J.Error.ExtraCode;

//Status_TF.ModAsse_K.Cmd					:= ModuloAsse_K.CmdExe.Code;
//Status_TF.ModAsse_K.CmdCase				:= ModuloAsse_K.CmdExe.CmdCase;
Status_TF.ModAsse_K.Error       		:= 0;//ModuloAsse_K.Error.Code;
Status_TF.ModAsse_K.ErrorExtra      	:= 0;//ModuloAsse_K.Error.ExtraCode;

//Status_TF.ModAspirazione.Cmd			:= ModuloAspirazione.CmdExe.Code;
//Status_TF.ModAspirazione.CmdCase		:= ModuloAspirazione.CmdExe.CmdCase;
Status_TF.ModAspirazione.Error       	:= MachinePalletizerModules.Pinza.Error.Code;
Status_TF.ModAspirazione.ErrorExtra     := MachinePalletizerModules.Pinza.Error.ExtraCode;

Status_TF.Pinza.Module.Error       	:= MachinePalletizerModules.Pinza.Error.Code;
Status_TF.Pinza.Module.ErrorExtra     := MachinePalletizerModules.Pinza.Error.ExtraCode;


(* Trsferimento a Struttura dati Creo *)
Status.MachineAuto := Status_TF.Macchina.Auto;
Status.MachineError := Status_TF.Macchina.Error;
Status.MachineErrorExtra := Status_TF.Macchina.ErrorExtra;

//Pinza Cilindro Cilindro Aspirazione DX
Status_TF.Pinza.AspirazioneDX.Active 			:= MachinePalletizerModules.Pinza.AspirazioneDX1^.Status.Aspirazione_ON; 
Status_TF.Pinza.AspirazioneDX.Inactive 		:= MachinePalletizerModules.Pinza.AspirazioneDX1^.Status.Aspirazione_OFF; 
Status_TF.Pinza.AspirazioneDX.SensorActive 	:= MachinePalletizerModules.Pinza.AspirazioneDX1^.Status.DepressioneSoglia1_OK; 
Status_TF.Pinza.AspirazioneDX.SensorInactive 	:= NOT MachinePalletizerModules.Pinza.AspirazioneDX1^.Status.DepressioneSoglia1_OK; 

Status_TF.Pinza.AspirazioneDX.Error := ErrBASEOVEM+MachinePalletizerModules.Pinza.AspirazioneDX1^.Status.ErrorID;
IF Status_TF.Pinza.AspirazioneDX.Error <> ErrBASEOVEM THEN 
	Status_TF.Pinza.AspirazioneDX.StatusToHMI := 9;
ELSIF MachinePalletizerModules.Pinza.AspirazioneDX1^.Status.Aspirazione_ON THEN
	Status_TF.Pinza.AspirazioneDX.StatusToHMI := 1;
ELSIF MachinePalletizerModules.Pinza.AspirazioneDX1^.Status.Aspirazione_OFF THEN
	Status_TF.Pinza.AspirazioneDX.StatusToHMI := 2;
END_IF
IF Status_TF.Pinza.AspirazioneDX.Error = ErrBASEOVEM THEN
	Status_TF.Pinza.AspirazioneDX.Error := 0;
END_IF


//Pinza Cilindro Cilindro AspirazioneFalda SX
Status_TF.Pinza.AspirazioneSX.Active 			:= MachinePalletizerModules.Pinza.AspirazioneSX1^.Status.Aspirazione_ON; 
Status_TF.Pinza.AspirazioneSX.Inactive 		:= MachinePalletizerModules.Pinza.AspirazioneSX1^.Status.Aspirazione_OFF; 
Status_TF.Pinza.AspirazioneSX.SensorActive 	:= MachinePalletizerModules.Pinza.AspirazioneSX1^.Status.DepressioneSoglia1_OK; 
Status_TF.Pinza.AspirazioneSX.SensorInactive 	:= NOT MachinePalletizerModules.Pinza.AspirazioneSX1^.Status.DepressioneSoglia1_OK; 

Status_TF.Pinza.AspirazioneSX.Error := ErrBASEOVEM+MachinePalletizerModules.Pinza.AspirazioneSX1^.Status.ErrorID ;
IF Status_TF.Pinza.AspirazioneSX.Error  <> ErrBASEOVEM THEN 
	Status_TF.Pinza.AspirazioneSX.StatusToHMI := 9;
ELSIF MachinePalletizerModules.Pinza.AspirazioneSX1^.Status.Aspirazione_ON THEN
	Status_TF.Pinza.AspirazioneSX.StatusToHMI := 1;
ELSIF MachinePalletizerModules.Pinza.AspirazioneSX1^.Status.Aspirazione_OFF THEN
	Status_TF.Pinza.AspirazioneSX.StatusToHMI := 2;
END_IF
IF Status_TF.Pinza.AspirazioneSX.Error = ErrBASEOVEM THEN
	Status_TF.Pinza.AspirazioneSX.Error := 0;
END_IF

//Pinza Cilindro Cilindro Apertura pinza 
Status_TF.Pinza.CilindroApertura.Active 			:= MachinePalletizerModules.Pinza.CilindroApertura^.Status.Active; 
Status_TF.Pinza.CilindroApertura.Inactive 			:= MachinePalletizerModules.Pinza.CilindroApertura^.Status.Inactive; 
Status_TF.Pinza.CilindroApertura.SensorActive 		:= MachinePalletizerModules.Pinza.CilindroApertura^.IN.PX_Active; 
Status_TF.Pinza.CilindroApertura.SensorInactive 	:= NOT MachinePalletizerModules.Pinza.CilindroApertura^.IN.PX_Inactive; 

Status_TF.Pinza.CilindroApertura.Error := MachinePalletizerModules.Pinza.CilindroApertura^.Status.ErrorID ;
IF Status_TF.Pinza.CilindroApertura.Error  <> 0 THEN 
	Status_TF.Pinza.CilindroApertura.StatusToHMI := 9;
ELSIF MachinePalletizerModules.Pinza.CilindroApertura^.Status.Active THEN
	Status_TF.Pinza.CilindroApertura.StatusToHMI := 1;
ELSIF MachinePalletizerModules.Pinza.CilindroApertura^.Status.Inactive THEN
	Status_TF.Pinza.CilindroApertura.StatusToHMI := 2;
END_IF
IF Status_TF.Pinza.CilindroApertura.Error = 0 THEN
	Status_TF.Pinza.CilindroApertura.Error := 0;
END_IF

//Aspirazione SX2 
Status_TF.Pinza.AspirazioneSX2.Active 			:= MachinePalletizerModules.Pinza.AspirazioneSX2^.Status.Aspirazione_ON; 
Status_TF.Pinza.AspirazioneSX2.Inactive 		:= MachinePalletizerModules.Pinza.AspirazioneSX2^.Status.Aspirazione_OFF; 
Status_TF.Pinza.AspirazioneSX2.SensorActive 	:= MachinePalletizerModules.Pinza.AspirazioneSX2^.Status.DepressioneSoglia1_OK; 
Status_TF.Pinza.AspirazioneSX2.SensorInactive 	:= NOT MachinePalletizerModules.Pinza.AspirazioneSX2^.Status.DepressioneSoglia1_OK; 

Status_TF.Pinza.AspirazioneSX2.Error := ErrBASEOVEM+MachinePalletizerModules.Pinza.AspirazioneSX2^.Status.ErrorID ;
IF Status_TF.Pinza.AspirazioneSX2.Error  <> ErrBASEOVEM THEN 
	Status_TF.Pinza.AspirazioneSX2.StatusToHMI := 9;
ELSIF MachinePalletizerModules.Pinza.AspirazioneSX2^.Status.Aspirazione_ON THEN
	Status_TF.Pinza.AspirazioneSX2.StatusToHMI := 1;
ELSIF MachinePalletizerModules.Pinza.AspirazioneSX2^.Status.Aspirazione_OFF THEN
	Status_TF.Pinza.AspirazioneSX2.StatusToHMI := 2;
END_IF
IF Status_TF.Pinza.AspirazioneSX2.Error = ErrBASEOVEM THEN
	Status_TF.Pinza.AspirazioneSX2.Error := 0;
END_IF
//Aspirazione DX 
Status_TF.Pinza.AspirazioneDX2.Active 			:= MachinePalletizerModules.Pinza.AspirazioneDX2^.Status.Aspirazione_ON; 
Status_TF.Pinza.AspirazioneDX2.Inactive 		:= MachinePalletizerModules.Pinza.AspirazioneDX2^.Status.Aspirazione_OFF; 
Status_TF.Pinza.AspirazioneDX2.SensorActive 	:= MachinePalletizerModules.Pinza.AspirazioneDX2^.Status.DepressioneSoglia1_OK; 
Status_TF.Pinza.AspirazioneDX2.SensorInactive 	:= NOT MachinePalletizerModules.Pinza.AspirazioneDX2^.Status.DepressioneSoglia1_OK; 

Status_TF.Pinza.AspirazioneDX2.Error := ErrBASEOVEM+MachinePalletizerModules.Pinza.AspirazioneDX2^.Status.ErrorID;
IF Status_TF.Pinza.AspirazioneDX2.Error <> ErrBASEOVEM THEN 
	Status_TF.Pinza.AspirazioneDX2.StatusToHMI := 9;
ELSIF MachinePalletizerModules.Pinza.AspirazioneDX2^.Status.Aspirazione_ON THEN
	Status_TF.Pinza.AspirazioneDX2.StatusToHMI := 1;
ELSIF MachinePalletizerModules.Pinza.AspirazioneDX2^.Status.Aspirazione_OFF THEN
	Status_TF.Pinza.AspirazioneDX2.StatusToHMI := 2;
END_IF
IF Status_TF.Pinza.AspirazioneDX.Error = ErrBASEOVEM THEN
	Status_TF.Pinza.AspirazioneDX.Error := 0;
END_IF

//Pinza Cilindro Cilindro Sblocco Rotazione
Status_TF.Pinza.CilindroSbloccoRotazione.Active 			:= MachinePalletizerModules.Pinza.CilindroSbloccoRotazione^.Status.Active; 
Status_TF.Pinza.CilindroSbloccoRotazione.Inactive 			:= MachinePalletizerModules.Pinza.CilindroSbloccoRotazione^.Status.Inactive; 
Status_TF.Pinza.CilindroSbloccoRotazione.SensorActive 		:= MachinePalletizerModules.Pinza.CilindroSbloccoRotazione^.IN.PX_Active; 
Status_TF.Pinza.CilindroSbloccoRotazione.SensorInactive 	:= NOT MachinePalletizerModules.Pinza.CilindroSbloccoRotazione^.IN.PX_Inactive; 

Status_TF.Pinza.CilindroSbloccoRotazione.Error := MachinePalletizerModules.Pinza.CilindroSbloccoRotazione^.Status.ErrorID ;
IF Status_TF.Pinza.CilindroSbloccoRotazione.Error  <> 0 THEN 
	Status_TF.Pinza.CilindroSbloccoRotazione.StatusToHMI := 9;
ELSIF MachinePalletizerModules.Pinza.CilindroSbloccoRotazione^.Status.Active THEN
	Status_TF.Pinza.CilindroSbloccoRotazione.StatusToHMI := 1;
ELSIF MachinePalletizerModules.Pinza.CilindroSbloccoRotazione^.Status.Inactive THEN
	Status_TF.Pinza.CilindroSbloccoRotazione.StatusToHMI := 2;
END_IF
IF Status_TF.Pinza.CilindroSbloccoRotazione.Error = 0 THEN
	Status_TF.Pinza.CilindroSbloccoRotazione.Error := 0;
END_IF

//Pinza Cilindro Cilindro Sblocco Bascolante
Status_TF.Pinza.CilindroSbloccoBascolante.Active 			:= MachinePalletizerModules.Pinza.CilindroSbloccoBascolante^.Status.Active; 
Status_TF.Pinza.CilindroSbloccoBascolante.Inactive 			:= MachinePalletizerModules.Pinza.CilindroSbloccoBascolante^.Status.Inactive; 
Status_TF.Pinza.CilindroSbloccoBascolante.SensorActive 		:= MachinePalletizerModules.Pinza.CilindroSbloccoBascolante^.IN.PX_Active; 
Status_TF.Pinza.CilindroSbloccoBascolante.SensorInactive 	:= NOT MachinePalletizerModules.Pinza.CilindroSbloccoBascolante^.IN.PX_Inactive; 

Status_TF.Pinza.CilindroSbloccoBascolante.Error := MachinePalletizerModules.Pinza.CilindroSbloccoBascolante^.Status.ErrorID ;
IF Status_TF.Pinza.CilindroSbloccoBascolante.Error  <> 0 THEN 
	Status_TF.Pinza.CilindroSbloccoBascolante.StatusToHMI := 9;
ELSIF MachinePalletizerModules.Pinza.CilindroSbloccoBascolante^.Status.Active THEN
	Status_TF.Pinza.CilindroSbloccoBascolante.StatusToHMI := 1;
ELSIF MachinePalletizerModules.Pinza.CilindroSbloccoBascolante^.Status.Inactive THEN
	Status_TF.Pinza.CilindroSbloccoBascolante.StatusToHMI := 2;
END_IF
IF Status_TF.Pinza.CilindroSbloccoBascolante.Error = 0 THEN
	Status_TF.Pinza.CilindroSbloccoBascolante.Error := 0;
END_IF


//Trasferisco segnalazione stato a HMI
IF Mission.State > 0 THEN
	StatoMissione := Mission.State;
ELSE
	StatoMissione := MISSION_STATE_NOP;
END_IF
//Aggiorno valori stato postazione
FOR i:=1 TO MAXAREAPRESENT DO
	HMI_Stato_Postazione[i].Abilitata 			:= WorkArea[i].Enable; 
	HMI_Stato_Postazione[i].CodiceFormatura		:= WorkAreaState[i].F;
	HMI_Stato_Postazione[i].CodiceLavorazione	:= WorkAreaState[i].Code;
	HMI_Stato_Postazione[i].LGV_Req				:= WorkAreaState[i].LGV_Req;
	HMI_Stato_Postazione[i].NPezzi				:= WorkAreaState[i].P -1;
	HMI_Stato_Postazione[i].ProgressiveNr		:= TO_UDINT(WorkAreaState[i].ID);	
	HMI_Stato_Postazione[i].Stato 				:= WorkAreaState[i].State;
	HMI_Stato_Postazione[i].TipologiaPostazione := WorkArea[i].Typology;
	HMI_Stato_Postazione[i].TipologiaSupporto 	:= WorkAreaState[i].Supporto.Tipologia;
	IF Status_TF.Macchina.Auto THEN
		HMI_NumeroPezziPresentiPostazione[i] := MAX(0,WorkAreaState[i].P-1);
		IF WorkAreaState[i].Supporto.Tipologia = CAVALLETTO THEN 
			HMI_NumeroPezziPresentiCavallete[i].HMI_NumeroPezziPresentiPostazione_A_Cavaleto := MAX(0,WorkAreaState[i].P_Cava.HMI_NumeroPezziPresentiPostazione_A_Cavaleto-1);
			HMI_NumeroPezziPresentiCavallete[i].HMI_NumeroPezziPresentiPostazione_B_Cavaleto := MAX(0,WorkAreaState[i].P_Cava.HMI_NumeroPezziPresentiPostazione_B_Cavaleto-1);
		END_IF
		
	END_IF
END_FOR

//STATO SICUREZZE
HMI_Status_FungiPal_OK 			:= I_SafetyStateEmergenza_PS306_307 = 1 AND I_SafetyStateEmergenza_PS308_309 = 1;
HMI_Status_FungoGenerale_OK 	:= I_SafetyStateEmergenze_Generali = 1;
HMI_Status_Funghi_OK 			:= HMI_Status_FungiPal_OK AND
                                   HMI_Status_FungoGenerale_OK;
 	    
HMI_Status_BarrierDXPal_OK 			:= I_SafetyStateBarrierDXPal  = 1;	
HMI_Status_BarrierSXPal_OK 			:= I_SafetyStateBarrierSXPal  = 1;				
HMI_Status_BarrierCentroDXPal_OK	:= I_SafetyStateBarrierCentroDXPal  = 1;		
HMI_Status_BarrierCentroSXPal_OK	:= I_SafetyStateBarrierCentroSXPal  = 1;		
HMI_Status_StateBarrierKarv_OK    	:= I_SafetyStateBarrierKarv  = 1;				

HMI_Status_BarrieraPall_OK			:= HMI_Status_BarrierDXPal_OK AND 		   
                                       HMI_Status_BarrierSXPal_OK AND 		   
                                       HMI_Status_BarrierCentroDXPal_OK AND
                                       HMI_Status_BarrierCentroSXPal_OK AND
									   HMI_Status_StateBarrierKarv_OK;
(*VISUALIZZAZIONE I/O SU PREMIUM HMI*)
HMI_AP200_2 := I_AP200_2;  	
HMI_AP200_3 := I_AP200_3;  
HMI_AP200_4 := I_AP200_4;  
HMI_AP200_5 := I_AP200_5;  
HMI_AP200_6	:= I_AP200_6;	 
HMI_AP200_7	:= I_AP200_7;	 
HMI_AP200_8 := I_AP200_8;  
HMI_AP200_9	:= I_AP200_9;	 
HMI_AP200_10:= I_AP200_10; 
HMI_AP201_2	:= I_AP201_2;	 
HMI_AP201_4 := O_AP201_4;  
HMI_AP201_5	:= I_AP201_5;	 
HMI_AP201_6 := O_AP201_6;  
HMI_AP201_3 := I_AP201_3;  
HMI_AP202_2	:= I_AP202_2;	 
HMI_AP202_3	:= I_AP202_3;	 
HMI_AP202_5	:= I_AP202_5;	 
HMI_AP202_6	:= I_AP202_6;	 

HMI_DepressioneOVEM_DX1 := Pinza.Ovem1.Status.ValoreDepressioneIstantanea;
HMI_DepressioneOVEM_DX2 := Pinza.Ovem12.Status.ValoreDepressioneIstantanea;

HMI_DepressioneOVEM_SX1 := Pinza.Ovem2.Status.ValoreDepressioneIstantanea;
HMI_DepressioneOVEM_SX2 := Pinza.Ovem22.Status.ValoreDepressioneIstantanea;

{info 'TODO:SISTEMARE IO PINZA X HMI'}	
//HMI_DepressioneOVEM_SX1 
////
//HMI_LetturaFTCPinza0_1 	
//HMI_LetturaFTCPinza180_1
//HMI_DepressioneOVEM_SX2 
////CIABATTA 516	
//HMI_DepressioneOVEM_DX1 
//HMI_DepressioneOVEM_DX2 
//HMI_LetturaFTCPinza0_2	
//HMI_LetturaFTCPinza180_2
//HMI_K516_51 			
//HMI_K516_52 			
//HMI_K516_61 			
//HMI_K516_62 			
//HMI_K516_71 			
//HMI_K516_72 			
//HMI_K516_81 			
//HMI_K516_82 			
////CIABATTA 517	
//HMI_K517_11  			
//HMI_K517_12  			
//HMI_K517_21  			
//HMI_K517_22  			
//HMI_K517_31  			
//HMI_K517_32  			
//HMI_K517_41  			
//HMI_K517_42  			
//HMI_K517_51 			
//HMI_K517_52 			
//HMI_K517_61 			
//HMI_K517_62 			
//HMI_K517_71 			
//HMI_K517_72 			
//HMI_K517_81 			
//HMI_K517_82
END_ACTION

ACTION _08_DataLogger_ACT:
// INIT - Assegnazione codici in verifica da formature - Verifico su quale fomatura è associato l codice i-esimo e scrivo la formatura associata nell'array di riferimento.
// Non posso avere duplicazioni in quanto è il supervisore a verificare che tutto sia concorde
// L'Array ottenuto, rappresenta la sequenza delle formature in cui ho un codice i-esimo
// es: formatura 1 con codici assegnati 7 e 10, formatura 3 con codicie da 1 a 4 pieni e formatura 4 con codice 15 -> 3,3,3,3,0,0,1,0,0,1,0,0,0,0,4.....
// Step 1 - cancello struttura
FOR k := 1 TO MAXFORMINGCODE DO
	DATA_LOGGER.Formign_ID_Active_Code[k] := 0;
END_FOR
// Step 2 - assegno valori attuali
FOR i := 1 TO MAXFORMING DO
	FOR k := 1 TO MAXFORMINGCODE DO 
		IF Forming[i].Code[k] <> 0 and Forming[i].Code[k] <> -1 THEN
			DATA_LOGGER.Formign_ID_Active_Code[k] := UINT_TO_INT(i);
		END_IF
	END_FOR
END_FOR

DLogger(Auto_GENERAL :=  MachinePalletizer_TF.CmdExe.Code = CmdDO, 
		Alarm_GENERAL := MachinePalletizer_TF.OUT.Error AND MachinePalletizer_TF.CmdExe.Code <> CmdDO,Man_GENERAL := MachinePalletizer_TF.IN.Mode.Man AND Status.MachineError = 0, 
		RI_GENERAL := MachinePalletizerGatesAccess.GateAccessConsolle.AccesActive (*OR MachinePalletizerGatesAccess.GateAccess2.AccesActive*),// OR MachinePalletizerLGV.LGVAccesActive, 
		Global_Reset := DLOG_Cmd_ResetCounter, 
		Daily_Reset := INT_TO_WORD(DLOG_Day_Reset), Weekly_Reset := INT_TO_WORD(DLOG_Week_Reset),
		Alarm_Reset := DLOG_Cmd_Alarm_reset,
		StoricoFile := DLOG_SaveDataOnReset,
		FilePath := 'C:\Logger\LogFile.txt',
		Channel := Channels);
		
Clogger(Global_Reset := CLOG_Global_reset,
		Daily_Reset := INT_TO_WORD(DLOG_Day_Reset), Weekly_Reset := INT_TO_WORD(DLOG_Week_Reset),
		Alarm_Reset := DLOG_Cmd_Alarm_reset,
		StoricoFile := DLOG_SaveDataOnReset,
		FilePath := 'C:\Logger\LogCounter.txt',
		Enable_Log_HMI := dlogger.Enable_Log_HMI,
		NumeroCanaliDatiProd := 16,
		Channel := Counters);
		
// Impostazione canali DataLogger
// Canale 1 - Mancanza pallet vuoti in ciclo automatico
Channels[0].Enable := TRUE;
Channels[0].Nome := 'Mancanza pallet vuoti in ciclo automatico';
Channels[0].Signal := PalletStackEmpty = 1 AND MachinePalletizer_TF.WorkAreaManager^.State = WAMANAGER_NOP AND MachinePalletizer_TF.CmdExe.Code = CmdDO;
Channels[0].Daily_Reference_Total := DLogger.Stat_Auto.Daily_Counter_State;
Channels[0].Weekly_Reference_Total := DLogger.Stat_Auto.Weekly_Counter_State;

// Canale 2 - Nessuna missione attiva su pallettizzatore in ciclo automatico
Channels[1].Enable := TRUE;
Channels[1].Nome := 'Nessuna missione attiva su pallettizzatore in ciclo automatico';
Channels[1].Signal := MachinePalletizer_TF.WorkAreaManager^.State = WAMANAGER_NOP AND MachinePalletizer_TF.CmdExe.Code = CmdDO;
Channels[1].Daily_Reference_Total := DLogger.Stat_Auto.Daily_Counter_State;
Channels[1].Weekly_Reference_Total := DLogger.Stat_Auto.Weekly_Counter_State;

// Canale 3 - Richiesta ingresso navetta su richiesta ingresso generale
(*Channels[2].Enable := TRUE;
Channels[2].Nome := 'Richiesta ingresso navetta su richiesta ingresso generale';
Channels[2].Signal := MachinePalletizerLGV.LGVAccesActive;
Channels[2].Daily_Reference_Total := DLogger.Stat_RI.Daily_Counter_State;
Channels[2].Weekly_Reference_Total := DLogger.Stat_RI.Weekly_Counter_State;
*)
// Canale 4 - Tutte le WA impegnate sul totale di automatico
Channels[3].Enable := TRUE;
Channels[3].Nome := 'Tutte le WA impegnate sul totale di automatico';
Channels[3].Signal := MachinePalletizer_TF.AllWABusy = 1 AND MachinePalletizer_TF.CmdExe.Code = CmdDO;
Channels[3].Daily_Reference_Total := DLogger.Stat_Auto.Daily_Counter_State;
Channels[3].Weekly_Reference_Total := DLogger.Stat_Auto.Weekly_Counter_State;

// Canale 5 - Tutte le WA impegnate sul totale di missione nulla
Channels[4].Enable := TRUE;
Channels[4].Nome := 'Tutte le WA impegnate sul totale di missione nulla';
Channels[4].Signal := MachinePalletizer_TF.AllWABusy = 1 AND MachinePalletizer_TF.CmdExe.Code = CmdDO;
Channels[4].Daily_Reference_Total := Channels[1].Daily_Counter_State;
Channels[4].Weekly_Reference_Total := Channels[1].Weekly_Counter_State;


////////////////////////////////////////////////////////////////////////////////////////////////////////
////////////////////////////////////////////////////////////////////////////////////////////////////////
// Impostazione canali CounterLogger
// Canale 1 - Totale pacchi prelevati - riservato non resettabile da operatore
Counters[0].Enable := TRUE;
Counters[0].Nome := 'Totale pacchi prelevati da ribaltino';
Counters[0].Signal := MachinePalletizer_TF.CmdExe.Code = CmdDO AND PaccoPresoXDataLogger;
Counters[0].Enable_Reset_Storico := FALSE;
Counters[0].ResetCounter := FALSE;
Counters[0].Daily_Reference_Total := 100;
Counters[0].Weekly_Reference_Total := 100;


// Canale 2 - Totale Pacchi parziali
Counters[1].Enable := TRUE;
Counters[1].Nome := 'Totale pacchi prelevati da ribaltino - parziale';
Counters[1].Signal := MachinePalletizer_TF.CmdExe.Code = CmdDO AND PaccoPresoXDataLogger;
Counters[1].Enable_Reset_Storico := FALSE;
Counters[1].ResetCounter := DATA_LOGGER.Reset_Operatore;
Counters[1].Daily_Reference_Total := 100;
Counters[1].Weekly_Reference_Total := 100;
Counters[1].Enable_Reset_Dopo_Salvataggio := TRUE;

(*
// Verifica segnale codice assegnato
FOR i := 1 TO 15 DO
	Counters[i + 1].Signal := MachinePalletizer_TF.CmdExe.Code = CmdDO AND PaccoPresoXDataLogger 
				AND WorkPickPointState[Mission.PPick].Code = (*Forming[DATA_LOGGER.Formign_ID_Active_Code[i]].Code[i]*) i AND WorkPickPointState[Mission.PPick].Code <> 0;
END_FOR
*)
// Conteggio riferimento pacchi parziali - somma di tutti i pacchi contati atualmente dopo reset parziale
TotalePacchiParziali := 0;
FOR i := 2 TO 16 DO
	TotalePacchiParziali := TotalePacchiParziali + Counters[I].Daily_Periodic_Counter_State;
END_FOR

// Canale 3 - Totale pacchi primo codice - parziale
Counters[2].Enable := TRUE;
Counters[2].Nome := CONCAT(STR1:= 'Primo codice - parziale, VALORE -> ', STR2 := INT_TO_STRING(1));
Counters[2].Enable_Reset_Storico := FALSE;
Counters[2].ResetCounter := DATA_LOGGER.Reset_Operatore;
Counters[2].Daily_Reference_Total := Counters[1].Daily_Counter_State;
Counters[2].Weekly_Reference_Total := Counters[1].Weekly_Counter_State;
Counters[2].Periodic_Reference_Total := TotalePacchiParziali;
Counters[2].Enable_Reset_Dopo_Salvataggio := TRUE;

// Canale 3 - Totale pacchi secondo codice - parziale
Counters[3].Enable := TRUE;
Counters[3].Nome := CONCAT(STR1:= 'Secondo codice - parziale, VALORE -> ', STR2 := INT_TO_STRING(2));
Counters[3].Enable_Reset_Storico := FALSE;
Counters[3].ResetCounter := DATA_LOGGER.Reset_Operatore;
Counters[3].Daily_Reference_Total := Counters[1].Daily_Counter_State;
Counters[3].Weekly_Reference_Total := Counters[1].Weekly_Counter_State;
Counters[3].Periodic_Reference_Total := TotalePacchiParziali;
Counters[3].Enable_Reset_Dopo_Salvataggio := TRUE;

// Canale 4 - Totale pacchi terzo codice - parziale
Counters[4].Enable := TRUE;
Counters[4].Nome := CONCAT(STR1:= 'Terzo codice - parziale, VALORE -> ', STR2 := INT_TO_STRING(3));
Counters[4].Enable_Reset_Storico := FALSE;
Counters[4].ResetCounter := DATA_LOGGER.Reset_Operatore;
Counters[4].Daily_Reference_Total := Counters[1].Daily_Counter_State;
Counters[4].Weekly_Reference_Total := Counters[1].Weekly_Counter_State;
Counters[4].Periodic_Reference_Total := TotalePacchiParziali;
Counters[4].Enable_Reset_Dopo_Salvataggio := TRUE;

// Canale 5 - Totale pacchi quarto codice - parziale
Counters[5].Enable := TRUE;
Counters[5].Nome := CONCAT(STR1:= 'Quarto codice - parziale, VALORE -> ', STR2 := INT_TO_STRING(4));
Counters[5].Enable_Reset_Storico := FALSE;
Counters[5].ResetCounter := DATA_LOGGER.Reset_Operatore;
Counters[5].Daily_Reference_Total := Counters[1].Daily_Counter_State;
Counters[5].Weekly_Reference_Total := Counters[1].Weekly_Counter_State;
Counters[5].Periodic_Reference_Total := TotalePacchiParziali;
Counters[5].Enable_Reset_Dopo_Salvataggio := TRUE;

